(* PLC project TC3_TE1400_GeneratedModule_train_anarx_FB, Beckhoff Automation GmbH & Co. KG TwinCAT 3 Function - TE1400 1.2.1240 *)
(* stored: companyURL www.beckhoff.com, creationDateTime 2022-07-14T09:12:33 *)

TYPE E_TcMatSimDataAreaType : (NotSpecified := 0, Standard, InputSrc, InputDst, OutputSrc, OutputDst, InternalDa, MArea, RetainDa);
END_TYPE

TYPE ST_TcMatSimObjectDataAreaInfo : STRUCT
  pPlcVar : PVOID;
  pModuleProcImg : PVOID;
  nSize : UDINT;
  nDataAreaId : UDINT;
  eDataAreaType : E_TcMatSimDataAreaType;
END_STRUCT;
END_TYPE

{attribute 'pack_mode' := '4'}
TYPE ST_train_anarxInitData : STRUCT
  Header : TComInitDataHdr;
  CallByHdr : TComInitDataElmHdr;
  CallBy : TctModuleCallByType;
  ExecutionSequenceHdr : TComInitDataElmHdr;
  ExecutionSequence : TctModuleExecutionSequenceType;
  StepSizeHdr : TComInitDataElmHdr;
  StepSize : TctStepSizeType;
  ExtendedFileAccessOIDHdr : TComInitDataElmHdr;
  ExtendedFileAccessOID : OTCID;
  ExecuteModelCodeHdr : TComInitDataElmHdr;
  ExecuteModelCode : BOOL;
  ModelParametersHdr : TComInitDataElmHdr;
  ModelParameters : P_train_anarx_T;
  ContextInfoArr_0_TaskOidHdr : TComInitDataElmHdr;
  ContextInfoArr_0_TaskOid : OTCID;
  ContextInfoArr_0_TaskPriorityHdr : TComInitDataElmHdr;
  ContextInfoArr_0_TaskPriority : UDINT;
  ContextInfoArr_0_TaskCycleTimeNsHdr : TComInitDataElmHdr;
  ContextInfoArr_0_TaskCycleTimeNs : UDINT;
  ContextInfoArr_0_TaskPortHdr : TComInitDataElmHdr;
  ContextInfoArr_0_TaskPort : UINT;
  ContextInfoArr_0_TaskSortOrderHdr : TComInitDataElmHdr;
  ContextInfoArr_0_TaskSortOrder : UDINT;
END_STRUCT;
END_TYPE

TYPE ST_train_anarx_Input : STRUCT
  Position_Increments : UDINT;
  Velocity_Increments : LREAL;
  DMS : DINT;
  actual_torque : INT;
END_STRUCT;
END_TYPE

TYPE ST_train_anarx_Output : STRUCT
  Control_Word : UINT;
  Target_Torque : INT;
  trigger : USINT;
  StartMeasurement : BOOL;
END_STRUCT;
END_TYPE

FUNCTION_BLOCK FB_TcMatSimObject
  VAR_INPUT
    bWriteFbInputValues : BOOL := TRUE;  (* set this flag to write FB input values to the TcComObject's input DataAreas. This will overwrite the mapped input values before module execution. Set to FALSE to read the mapped input values from the TcComObject to the FB. *)
  END_VAR
  VAR
    pDataAreas : POINTER TO ST_TcMatSimObjectDataAreaInfo;  (* process image src and dst pointers and sizes *)
    nDataAreas : UDINT;
    ipObjSrv : ITComObjectServer;  (* global interface pointers *)
    ipTcComObj : ITComObject;  (* object interface pointers *)
    ipTcCyclic : ITcCyclic;
    ipTcPostCyclic : ITcPostCyclic;
    ipTcAdi : ITcADI;
    ipTask : ITcTask;  (* task interface pointers *)
    pInitData : POINTER TO TComInitDataHdr;  (* initial parameters *)
    hResult : HRESULT;  (* hResult of interface calls (0 if no error) *)
    moduleClsId : CLSID;  (* module class ID *)
    assignedClsId : CLSID;  (* expected/desired module class ID *)
    bClassIdVerified : BOOL;
    bDynInstance : BOOL;  (* flag indicating whether the module instance was created dynamically *)
    eInitialObjState : TCOM_STATE := TCOM_STATE.TCOM_STATE_INIT;  (* the object state at the time FB_init was called, FB_exit will try to switch to this state (only if this means to shift down) *)
  END_VAR

            
          

{attribute 'object_name' := 'ReleaseTcComInterface'}
METHOD ReleaseTcComInterface : HRESULT
  VAR
    nStateChangeCnt : DINT := 0;
  END_VAR
                  
IF (ipTcComObj<>0) THEN
  WHILE (State>eInitialObjState AND nStateChangeCnt<1000) DO
    State := eInitialObjState;
    nStateChangeCnt := nStateChangeCnt+1;
  END_WHILE
  ReleaseObjInterfaces();
  IF (bDynInstance) THEN
    ReleaseTcComInterface := TC3_MODULE.FW_ObjMgr_DeleteInstance(ADR(ipTcComObj));
  ELSE
    ipTcComObj.TcRelease();
  END_IF
  ipTcComObj := 0;
END_IF
                  
                
END_METHOD

{attribute 'object_name' := 'ReleaseObjInterfaces'}
METHOD ReleaseObjInterfaces : HRESULT
                  
// release interface pointers
IF (ipTcCyclic<>0) THEN
  ipTcCyclic.TcRelease();
  ipTcCyclic := 0;
END_IF
IF (ipTcPostCyclic<>0) THEN
  ipTcPostCyclic.TcRelease();
  ipTcPostCyclic := 0;
END_IF
IF (ipTcAdi<>0) THEN
  ipTcAdi.TcRelease();
  ipTcAdi := 0;
END_IF
                  
                
END_METHOD

{attribute 'object_name' := 'Internal_SetObjState'}
METHOD Internal_SetObjState
  VAR_INPUT
    hr : REFERENCE TO HRESULT;
    nextState : TCOM_STATE;
  END_VAR
                  
// verify class id
IF (SUCCEEDED(hr)) THEN
  hr := VerifyClassId();
END_IF

// switch object state
IF (SUCCEEDED(hr) AND nextState>=TCOM_STATE_INIT) THEN
  IF (ipTcComObj=0) THEN
    hr := Tc2_System.E_HRESULTAdsErr.NOINTERFACE;
  END_IF
  IF (ipObjSrv=0) THEN
    hr := Tc2_System.E_HRESULTAdsErr.NOINTERFACE;
  END_IF
  IF (SUCCEEDED(hr)) THEN
    hr := ipTcComObj.TcSetObjState(nextState,ipObjSrv,pInitData);
  END_IF
END_IF
                  
                
END_METHOD

{attribute 'object_name' := 'FB_init'}
METHOD FB_init : BOOL
  VAR_INPUT
    bInitRetains : BOOL;  (* init retain variables *)
    bInCopyCode : BOOL;  (* Online Change *)
    oid : OTCID;
  END_VAR
                  
FB_init := SUCCEEDED(Init(oid));
                  
                
END_METHOD

{attribute 'object_name' := 'GetObjPara'}
METHOD GetObjPara : HRESULT
  VAR_INPUT
    pid : PTCID;
    nData : UDINT;
    pData : PVOID;
  END_VAR
                  
IF (ipTcComObj=0) THEN
  GetObjPara := Tc2_System.E_HRESULTAdsErr.NOINTERFACE;
END_IF

IF (SUCCEEDED(GetObjPara)) THEN
  GetObjPara := ipTcComObj.TcGetObjPara(pid:=pid,nData,pData,0);
END_IF
                  
                
END_METHOD

{attribute 'object_name' := 'QueryObjInterface'}
METHOD QueryObjInterface
  VAR_INPUT
    hr : REFERENCE TO HRESULT;
    iid : REFERENCE TO IID;
    pipItf : POINTER TO ITcUnknown;
  END_VAR
  VAR CONSTANT
    pNull : PVOID := 0;
  END_VAR
                  
IF (SUCCEEDED(hr)) THEN
  IF (ipTcComObj=0) THEN
    hr := Tc2_System.E_HRESULTAdsErr.NOINTERFACE;
  ELSIF (pipItf^=ULINT_TO_DWORD(pNull)) THEN
    hr := ipTcComObj.TcQueryInterface(iid:= iid, pipItf:=pipItf);
  END_IF
END_IF
                  
                
END_METHOD

{attribute 'object_name' := 'SaveOnlineParametersForInit'}
METHOD SaveOnlineParametersForInit : HRESULT
  VAR
    idx : UINT;
    pInitElemHdr : POINTER TO TComInitDataElmHdr;
    pData : PVOID;
    nData : UDINT;
  END_VAR
  VAR CONSTANT
    nInitDataAlignment : UDINT := 4;
  END_VAR
                  IF (pInitData<>0) THEN
  pInitElemHdr := pInitData + SIZEOF(pInitData^);
  FOR idx:=1 TO pInitData^.uiElmCnt DO
    pData := pInitElemHdr + ULINT_TO_DWORD(SIZEOF(pInitElemHdr^));
    nData := pInitElemHdr^.cbData;
    SaveOnlineParametersForInit := GetObjPara(pInitElemHdr^.indexOffset,nData,pData);
    IF (FAILED(SaveOnlineParametersForInit)) THEN
      RETURN;
    END_IF
    pInitElemHdr := pData + (nInitDataAlignment*((nData + nInitDataAlignment - 1)/nInitDataAlignment));
  END_FOR
ELSE
	SaveOnlineParametersForInit := Tc2_System.E_HRESULTAdsErr.NOTINIT;
END_IF
                  
                
END_METHOD

{attribute 'object_name' := 'ResetHresult'}
METHOD ResetHresult
                  hResult := S_OK;
                
END_METHOD

{attribute 'object_name' := 'Execute'}
METHOD Execute : HRESULT
  VAR
    nDaIdx : UDINT;
    pCurDataArea : POINTER TO ST_TcMatSimObjectDataAreaInfo;
  END_VAR
                  
IF (SUCCEEDED(hResult)) THEN
  hResult := VerifyClassId();
END_IF

IF (SUCCEEDED(hResult) AND State<>TCOM_STATE_OP) THEN
  hResult := Tc2_System.E_HRESULTAdsErr.NOTREADY;
END_IF

// get image pointers
IF (SUCCEEDED(hResult)) THEN
  GetImagePtrs(hResult);
END_IF

// copy inputs
IF (pDataAreas<>0 AND nDataAreas>0 AND bWriteFbInputValues) THEN
  FOR nDaIdx:=0 TO nDataAreas-1 DO
    IF (FAILED(hResult))THEN
      CONTINUE;
    END_IF
    pCurDataArea := pDataAreas + nDaIdx*SIZEOF(ST_TcMatSimObjectDataAreaInfo);
    IF ((pCurDataArea^.eDataAreaType <> E_TcMatSimDataAreaType.InputDst))THEN
      CONTINUE;
    END_IF
    IF (pCurDataArea^.pModuleProcImg<>0 AND pCurDataArea^.pPlcVar<>0) THEN
      MEMCPY(pCurDataArea^.pModuleProcImg,pCurDataArea^.pPlcVar,pCurDataArea^.nSize);
    ELSE
      hResult := Tc2_System.E_HRESULTAdsErr.NOINTERFACE;
    END_IF
  END_FOR
END_IF

// call cycle update
IF (SUCCEEDED(hResult)) THEN
  IF (ipTcCyclic<>0) THEN
    hResult := ipTcCyclic.CycleUpdate(ipTask:= ipTask, ipCaller:= 0, context:= 0);
  ELSE
    hResult := Tc2_System.E_HRESULTAdsErr.NOINTERFACE;
  END_IF
END_IF

// copy outputs
IF (pDataAreas<>0 AND nDataAreas>0) THEN
  FOR nDaIdx:=0 TO nDataAreas-1 DO
    IF (FAILED(hResult))THEN
      CONTINUE;
    END_IF
    pCurDataArea := pDataAreas + nDaIdx*SIZEOF(ST_TcMatSimObjectDataAreaInfo);
    IF ((pCurDataArea^.eDataAreaType = E_TcMatSimDataAreaType.OutputSrc) OR NOT bWriteFbInputValues) THEN
      IF (pCurDataArea^.pModuleProcImg<>0 AND pCurDataArea^.pPlcVar<>0) THEN
        MEMCPY(pCurDataArea^.pPlcVar,pCurDataArea^.pModuleProcImg,pCurDataArea^.nSize);
      ELSE
        hResult := Tc2_System.E_HRESULTAdsErr.NOINTERFACE;
      END_IF
    END_IF
  END_FOR
END_IF


// call post cyclic update
IF (SUCCEEDED(hResult)) THEN
  IF (ipTcPostCyclic<>0) THEN
    hResult := ipTcPostCyclic.PostCyclicUpdate(ipTask:= 0, ipCaller:= 0, context:= 0);
  ELSE
    hResult := Tc2_System.E_HRESULTAdsErr.NOINTERFACE;
  END_IF
END_IF

ReleaseImagePtrs();

Execute := hResult;
                  
                
END_METHOD

{attribute 'object_name' := 'GetImagePtrs'}
METHOD GetImagePtrs
  VAR_INPUT
    hr : REFERENCE TO HRESULT;
  END_VAR
  VAR
    nDaIdx : UDINT;
    pCurDataArea : POINTER TO ST_TcMatSimObjectDataAreaInfo;
  END_VAR
                  
IF (ipTcAdi=0) THEN
  hr := Tc2_System.E_HRESULTAdsErr.NOINTERFACE;
END_IF
IF(State<>TCOM_STATE_OP)THEN
  hr := Tc2_System.E_HRESULTAdsErr.INVALIDSTATE;
END_IF


// get pointers to process images
IF (pDataAreas<>0 AND nDataAreas>0) THEN
  FOR nDaIdx:=0 TO nDataAreas-1 DO
    pCurDataArea := pDataAreas + nDaIdx*SIZEOF(ST_TcMatSimObjectDataAreaInfo);
    IF (FAILED(hr))THEN
      CONTINUE;
    END_IF
    IF ((pCurDataArea^.eDataAreaType <> E_TcMatSimDataAreaType.InputDst) AND (pCurDataArea^.eDataAreaType <> E_TcMatSimDataAreaType.OutputSrc))THEN
      CONTINUE;
    END_IF
    IF (pCurDataArea^.pModuleProcImg=0 AND pCurDataArea^.nSize>0) THEN
      hr := ipTcAdi.GetImagePtr(size:= pCurDataArea^.nSize , offs:=0 , adi_x:=pCurDataArea^.nDataAreaId , ppData:=ADR(pCurDataArea^.pModuleProcImg));
    END_IF
  END_FOR
END_IF

IF (FAILED(hr)) THEN
  ReleaseImagePtrs();
END_IF
                  
                
END_METHOD

{attribute 'object_name' := 'VerifyClassId'}
METHOD VerifyClassId : HRESULT
  VAR
    emptyClsId : CLSID;
  END_VAR
                  memset(ADR(emptyClsId),0,SIZEOF(emptyClsId));
IF (bClassIdVerified) THEN
  // class ID was already verified
  VerifyClassId := Tc2_System.E_HRESULTAdsErr.HRESULT_ADS_NOERROR;
ELSIF (memcmp(ADR(assignedClsId),ADR(emptyClsId),SIZEOF(assignedClsId))=0) THEN
  // skip class ID verification if no assignedClsId specified
  VerifyClassId := Tc2_System.E_HRESULTAdsErr.HRESULT_ADS_NOERROR;
ELSE
  // verify class ID
  VerifyClassId := ReadModuleClassId();

  IF (SUCCEEDED(VerifyClassId)) THEN
    IF (memcmp(ADR(assignedClsId),ADR(moduleClsId),SIZEOF(assignedClsId))<>0) THEN
     VerifyClassId := Tc2_System.E_HRESULTAdsErr.INVALIDCLSID;
    END_IF
  END_IF
  bClassIdVerified := SUCCEEDED(VerifyClassId);
END_IF
                  
                
END_METHOD

{attribute 'object_name' := 'SetObjPara'}
METHOD SetObjPara : HRESULT
  VAR_INPUT
    pid : PTCID;
    nData : UDINT;
    pData : PVOID;
  END_VAR
                  
IF (ipTcComObj=0) THEN
  SetObjPara := Tc2_System.E_HRESULTAdsErr.NOINTERFACE;
END_IF

IF (SUCCEEDED(SetObjPara)) THEN
  SetObjPara := ipTcComObj.TcSetObjPara(pid:=pid,nData,pData,0);
END_IF
                  
                
END_METHOD

{attribute 'object_name' := 'QueryTcComInterface'}
METHOD QueryTcComInterface
  VAR_INPUT
    hr : REFERENCE TO HRESULT;
    oid : OTCID;
  END_VAR
                  
IF (ipObjSrv=0) THEN
  hr := Tc2_System.E_HRESULTAdsErr.NOINTERFACE;
END_IF

IF (SUCCEEDED(hr) AND ipTcComObj=0) THEN
  bDynInstance := FALSE;
  IF(oid>0) THEN
    // query interface of existing object
    hr := ipObjSrv.TcQueryObjectInterface(oid,IID_ITComObject,ADR(ipTcComObj));
  ELSE
    // create new instance and get the object interface
    hr := ipObjSrv.TcCreateInstance(assignedClsId,IID_ITComObject,ADR(ipTcComObj));
    IF (SUCCEEDED(hr)) THEN
      bDynInstance := TRUE;
      hr := ipTcComObj.TcSetObjectId(OTCID_CreateNewId);
    END_IF
  END_IF
  IF (SUCCEEDED(hr)) THEN
    eInitialObjState := State;
  END_IF
END_IF
                  
                
END_METHOD

{attribute 'object_name' := 'ReleaseImagePtrs'}
METHOD ReleaseImagePtrs : HRESULT
  VAR
    nDaIdx : UDINT;
    pCurDataArea : POINTER TO ST_TcMatSimObjectDataAreaInfo;
  END_VAR
                  
IF (ipTcAdi=0) THEN
  ReleaseImagePtrs := Tc2_System.E_HRESULTAdsErr.NOINTERFACE;
END_IF

IF (SUCCEEDED(ReleaseImagePtrs) AND pDataAreas<>0 AND nDataAreas>0) THEN
  // release pointers to the simulink module process images
  FOR nDaIdx:=0 TO nDataAreas-1 DO
    pCurDataArea := pDataAreas + nDaIdx*SIZEOF(ST_TcMatSimObjectDataAreaInfo);

    IF (pCurDataArea^.pModuleProcImg<>0) THEN
      ipTcAdi.ReleaseImagePtr(pData:=pCurDataArea^.pModuleProcImg);
      pCurDataArea^.pModuleProcImg := 0;
    END_IF
  END_FOR
END_IF
                  
                
END_METHOD

{attribute 'object_name' := 'FB_exit'}
METHOD FB_exit : BOOL
  VAR_INPUT
    bInCopyCode : BOOL;  (* Online Change *)
  END_VAR
                  
IF (NOT bInCopyCode) THEN
  IF (ipObjSrv<>0) THEN
    ipObjSrv.TcRelease();
    ipObjSrv := 0;
  END_IF

  ReleaseTcComInterface();
END_IF
                  
                
END_METHOD

{attribute 'object_name' := 'InitObjName'}
METHOD InitObjName
  VAR_INPUT
    hr : REFERENCE TO HRESULT;
  END_VAR
  VAR
    objectName : STRING(255) := 'TcMatSimObject_PlcRtFbInstance';
    oid : OTCID;
  END_VAR
                  
IF (SUCCEEDED(hr)) THEN
  hr := ipTcComObj.TcGetObjectId(oid);
END_IF

IF (SUCCEEDED(hr) and bDynInstance) THEN
  objectName := TC2_STANDARD.CONCAT(objectName,'_');
  objectName := TC2_STANDARD.CONCAT(objectName,UDINT_TO_STRING(oid));
  hr := ipTcComObj.TcSetObjectName(ADR(objectName));
END_IF
                  
                
END_METHOD

{attribute 'object_name' := 'SetObjState'}
METHOD SetObjState : HRESULT
  VAR_INPUT
    finalState : TCOM_STATE;
  END_VAR
  VAR
    bShiftUp : BOOL;
    bShiftDown : BOOL;
    currentState : TCOM_STATE;
  END_VAR
                  
currentState := State;

bShiftUp := finalState>currentState;
bShiftDown := finalState<currentState;

// do not switch up on error
IF (FAILED(hresult)) THEN
  bShiftUp := FALSE;
END_IF
// reset existing error on switching down
IF (bShiftDown) THEN
  ResetHresult();
END_IF

// prepared state switch
CASE currentState OF
  TCOM_STATE_INIT:
    IF(bShiftUp) THEN
      QueryTcComInterface(hResult,0);
      Internal_SetObjState(hResult,TCOM_STATE.TCOM_STATE_PREOP);
      InitObjName(hResult);
    END_IF

  TCOM_STATE_PREOP:
    IF(bShiftUp) THEN
      Internal_SetObjState(hResult,TCOM_STATE.TCOM_STATE_SAFEOP);
      QueryObjInterfaces(hResult);
    ELSIF (bShiftDown) THEN
      Internal_SetObjState(hResult,TCOM_STATE.TCOM_STATE_INIT);
    END_IF

  TCOM_STATE_SAFEOP:
    IF(bShiftUp) THEN
      Internal_SetObjState(hResult,TCOM_STATE.TCOM_STATE_OP);
      QueryObjInterfaces(hResult);
    ELSIF (bShiftDown) THEN
      Internal_SetObjState(hResult,TCOM_STATE.TCOM_STATE_PREOP);
      ReleaseObjInterfaces();
    END_IF


  TCOM_STATE_OP:
    IF (bShiftDown) THEN
      Internal_SetObjState(hResult,TCOM_STATE.TCOM_STATE_SAFEOP);
    END_IF
END_CASE

SetObjState := hResult;
                  
                
END_METHOD

{attribute 'object_name' := 'QueryObjInterfaces'}
METHOD QueryObjInterfaces
  VAR_INPUT
    hr : REFERENCE TO HRESULT;
  END_VAR
                  
IF(State<TCOM_STATE_PREOP)THEN
  hr := Tc2_System.E_HRESULTAdsErr.INVALIDSTATE;
END_IF

//cyclic interface
QueryObjInterface(hr,IID_ITCCYCLIC,ADR(ipTcCyclic));
//post cyclic interface
QueryObjInterface(hr,IID_ITCPOSTCYCLIC,ADR(ipTcPostCyclic));
//adi interface
QueryObjInterface(hr,IID_ITcADI,ADR(ipTcAdi));
                  
                
END_METHOD

{attribute 'object_name' := 'Init'}
METHOD Init : HRESULT
  VAR_INPUT
    oid : OTCID;
  END_VAR
                  
// preinitialize variables
memset(ADR(moduleClsId),0,SIZEOF(moduleClsId));
bClassIdVerified := FALSE;
hResult := Tc2_System.E_HRESULTAdsErr.HRESULT_ADS_NOERROR;

// get object server
IF (ipObjSrv=0) THEN
  hResult := FW_ObjMgr_GetObjectServer(_AppInfo.ObjId,ADR(ipObjSrv));
END_IF

// try to get object interfaces
IF (SUCCEEDED(hresult)) THEN
  QueryTcComInterface(hResult,oid);
END_IF

// verify class id
IF (SUCCEEDED(hresult)) THEN
  hresult := VerifyClassId();
END_IF

// query interfaces, if the current state is higher than INIT
IF (SUCCEEDED(hresult) AND State>TCOM_STATE.TCOM_STATE_INIT) THEN
  QueryObjInterfaces(hResult);
END_IF

// return value
Init := hresult;
                  
                
END_METHOD

{attribute 'object_name' := 'ReadModuleClassId'}
METHOD ReadModuleClassId : HRESULT
  VAR
    emptyClsId : CLSID;
  END_VAR
                  memset(ADR(emptyClsId),0,SIZEOF(emptyClsId));
IF (memcmp(ADR(moduleClsId),ADR(emptyClsId),SIZEOF(moduleClsId))=0) THEN
  IF (ipTcComObj=0) THEN
    ReadModuleClassId := Tc2_System.E_HRESULTAdsErr.NOINTERFACE;
  END_IF

  //objectClsId := clsid;
  IF (SUCCEEDED(ReadModuleClassId)) THEN
    ReadModuleClassId := ipTcComObj.GetClassId(moduleClsId);
  END_IF
END_IF
                
END_METHOD

METHOD PUBLIC AssignClassId
VAR_INPUT
	clsId : CLSID;
END_VAR
                  assignedClsId := clsId;
bClassIdVerified := false;
                  
                
END_METHOD

PROPERTY Error : BOOL
GET
                    Error := FAILED(hResult);
                  
END_GET
END_PROPERTY

METHOD PUBLIC SetDataAreaInfo
VAR_INPUT
  pDataAreas: POINTER TO ST_TcMatSimObjectDataAreaInfo;
  nDataAreas: UDINT;
END_VAR
                  
THIS^.nDataAreas := nDataAreas;
THIS^.pDataAreas := pDataAreas;
                  
                
END_METHOD

METHOD PUBLIC SetInitDataInfo
VAR_INPUT
  pInitData : POINTER TO TComInitDataHdr;
END_VAR
                  this^.pInitData := pInitData;
                
END_METHOD

PROPERTY ClassId : CLSID
GET
                    hResult := ReadModuleClassId();
ClassId := moduleClsId;
                    
                  
END_GET
END_PROPERTY

PROPERTY State : TCOM_STATE
GET
  VAR
    hr : HRESULT := S_OK;
    eObjState : TCOM_STATE;
  END_VAR
                    
IF (ipTcComObj<>0) THEN
  hr := ipTcComObj.TcGetObjState(ADR(eObjState));
IF (FAILED(hr)) THEN
  eObjState := TCOM_STATE.TCOM_STATE_INIT;
END_IF
ELSE
  eObjState := TCOM_STATE.TCOM_STATE_INIT;
END_IF
State := eObjState;
                    
                  
END_GET
SET
                    SetObjState(State);
                  
END_SET
END_PROPERTY

PROPERTY ErrorCode : HRESULT
GET
                    ErrorCode := hResult;
                  
END_GET
END_PROPERTY
END_FUNCTION_BLOCK

{attribute 'TcDependOnClassFactory' := 'train_anarx'}
FUNCTION_BLOCK FB_train_anarx EXTENDS FB_TcMatSimObject
  VAR_INPUT
    stInput : ST_train_anarx_Input;
  END_VAR
  VAR_OUTPUT
    stOutput : ST_train_anarx_Output;
  END_VAR
  VAR
    stInitData : ST_train_anarxInitData;
    arrDataAreas : ARRAY[1..2] OF ST_TcMatSimObjectDataAreaInfo;
    bParametersVerified : BOOL;
  END_VAR

            
          

{attribute 'object_name' := 'Internal_SetObjState'}
METHOD Internal_SetObjState
  VAR_INPUT
    hr : REFERENCE TO HRESULT;
    nextState : TCOM_STATE;
  END_VAR
                  
// update pointer to InitData structure
SetInitDataInfo(ADR(stInitData));
// call base method
SUPER^.Internal_SetObjState(hr,nextState);
                  
                
END_METHOD

{attribute 'object_name' := 'SaveOnlineParametersForInit'}
METHOD SaveOnlineParametersForInit : HRESULT
  VAR
    idx : UINT;
    pInitElemHdr : POINTER TO TComInitDataElmHdr;
    pData : PVOID;
    nData : UDINT;
  END_VAR
  VAR CONSTANT
    nInitDataAlignment : UDINT := 4;
  END_VAR
                  
// update pointer to InitData structure
SetInitDataInfo(ADR(stInitData));
// call base method
SaveOnlineParametersForInit := SUPER^.SaveOnlineParametersForInit();
                  
                
END_METHOD

METHOD FB_init : BOOL
  VAR_INPUT
    bInitRetains : BOOL;  (* if TRUE, the retain variables are initialized (warm start / cold start) *)
    bInCopyCode : BOOL;  (* if TRUE, the instance afterwards gets moved into the copy code (online change) *)
    oid : OTCID;
  END_VAR
  VAR
    clsId : CLSID;
  END_VAR
                  
// initialize flags
bParametersVerified := false;
                    
// set module class id for compatibility check
clsId.Data1 := 16#ed2a66fb;
clsId.Data2 := 16#550e;
clsId.Data3 := 16#4b31;
clsId.Data4[0] := 16#b5;
clsId.Data4[1] := 16#1b;
clsId.Data4[2] := 16#1e;
clsId.Data4[3] := 16#91;
clsId.Data4[4] := 16#4f;
clsId.Data4[5] := 16#8f;
clsId.Data4[6] := 16#f7;
clsId.Data4[7] := 16#c0;

AssignClassId(clsId);
                    
// initialize InitData structure with default values              
stInitData.CallByHdr.indexGroup := 0;
stInitData.CallByHdr.indexOffset := 16#00000000;
stInitData.CallByHdr.cbData := SIZEOF(stInitData.CallBy);
stInitData.CallBy := TctModuleCallByType.CyclicTask;
stInitData.ExecutionSequenceHdr.indexGroup := 0;
stInitData.ExecutionSequenceHdr.indexOffset := 16#00000001;
stInitData.ExecutionSequenceHdr.cbData := SIZEOF(stInitData.ExecutionSequence);
stInitData.ExecutionSequence := TctModuleExecutionSequenceType.StateUpdateAfterOutputMapping;
stInitData.StepSizeHdr.indexGroup := 0;
stInitData.StepSizeHdr.indexOffset := 16#00000002;
stInitData.StepSizeHdr.cbData := SIZEOF(stInitData.StepSize);
stInitData.StepSize := TctStepSizeType.RequireMatchingTaskCycleTime;
stInitData.ExtendedFileAccessOIDHdr.indexGroup := 0;
stInitData.ExtendedFileAccessOIDHdr.indexOffset := 16#00000005;
stInitData.ExtendedFileAccessOIDHdr.cbData := SIZEOF(stInitData.ExtendedFileAccessOID);
stInitData.ExtendedFileAccessOID := 0;
stInitData.ExecuteModelCodeHdr.indexGroup := 0;
stInitData.ExecuteModelCodeHdr.indexOffset := 16#00000008;
stInitData.ExecuteModelCodeHdr.cbData := SIZEOF(stInitData.ExecuteModelCode);
stInitData.ExecuteModelCode := 1;
stInitData.ModelParametersHdr.indexGroup := 0;
stInitData.ModelParametersHdr.indexOffset := 16#83000000;
stInitData.ModelParametersHdr.cbData := SIZEOF(stInitData.ModelParameters);
stInitData.ModelParameters._R[0] := 0.10557324255439252;
stInitData.ModelParameters._R[1] := 0.37689728877712958;
stInitData.ModelParameters._R[2] := 0.82623132681154499;
stInitData.ModelParameters._R[3] := 0.80515070185744342;
stInitData.ModelParameters._R[4] := 0.28033408284883216;
stInitData.ModelParameters._R[5] := 0.20419454517375848;
stInitData.ModelParameters._R[6] := 0.29127318222485832;
stInitData.ModelParameters._R[7] := 0.25248459304526055;
stInitData.ModelParameters._R[8] := 0.85181877670829109;
stInitData.ModelParameters._R[9] := 0.26730813856504498;
stInitData.ModelParameters._R[10] := 0.85973341835764761;
stInitData.ModelParameters._R[11] := 0.48821150954772086;
stInitData.ModelParameters._R[12] := 0.66695764239898803;
stInitData.ModelParameters._R[13] := 0.76922255995861488;
stInitData.ModelParameters._R[14] := 0.45433723001590831;
stInitData.ModelParameters._R[15] := 0.36540629909774192;
stInitData.ModelParameters._R[16] := 0.18448083270146118;
stInitData.ModelParameters._R[17] := 0.70086782168457618;
stInitData.ModelParameters._R[18] := 0.76784685041686818;
stInitData.ModelParameters._R[19] := 0.56414679263598622;
stInitData.ModelParameters._R[20] := 0.58598712526380503;
stInitData.ModelParameters._R[21] := 0.61005066126219132;
stInitData.ModelParameters._R[22] := 0.19543577562249415;
stInitData.ModelParameters._R[23] := 0.64329142670086592;
stInitData.ModelParameters._R[24] := 0.58267310864706856;
stInitData.ModelParameters._R[25] := 0.79798332299322849;
stInitData.ModelParameters._R[26] := 0.33180383592093965;
stInitData.ModelParameters._R[27] := 0.98316309922904865;
stInitData.ModelParameters._R[28] := 0.61220339829755299;
stInitData.ModelParameters._R[29] := 0.37845979384680939;
stInitData.ModelParameters._R[30] := 0.26096574430972613;
stInitData.ModelParameters._R[31] := 0.98801891092854388;
stInitData.ModelParameters._R[32] := 0.88761571192799182;
stInitData.ModelParameters._R[33] := 0.49443727460454467;
stInitData.ModelParameters._R[34] := 0.96137766517165912;
stInitData.ModelParameters._R[35] := 0.75085204485352486;
stInitData.ModelParameters._R[36] := 0.66551284350087503;
stInitData.ModelParameters._R[37] := 0.56475841691778406;
stInitData.ModelParameters._R[38] := 0.67811270612970664;
stInitData.ModelParameters._R[39] := 0.73032933705708902;
stInitData.ModelParameters._R[40] := 0.9876927697421114;
stInitData.ModelParameters._R[41] := 0.17853778300790973;
stInitData.ModelParameters._R[42] := 0.2112881137503454;
stInitData.ModelParameters._R[43] := 0.22263422347063244;
stInitData.ModelParameters._R[44] := 0.22981152085528173;
stInitData.ModelParameters._R[45] := 0.58054172851801422;
stInitData.ModelParameters._R[46] := 0.13458174770618431;
stInitData.ModelParameters._R[47] := 0.41675382902513802;
stInitData.ModelParameters._R[48] := 0.37503426129121775;
stInitData.ModelParameters._R[49] := 0.61532742494748438;
stInitData.ModelParameters._R[50] := 0.58497592475358873;
stInitData.ModelParameters._R[51] := 0.57088276882443501;
stInitData.ModelParameters._R[52] := 0.83801882588390086;
stInitData.ModelParameters._R[53] := 0.46346631174006891;
stInitData.ModelParameters._R[54] := 0.95558082085154439;
stInitData.ModelParameters._R[55] := 0.35709928964954307;
stInitData.ModelParameters._R[56] := 0.29876036646169085;
stInitData.ModelParameters._R[57] := 0.48986379749351949;
stInitData.ModelParameters._R[58] := 0.24301356646415506;
stInitData.ModelParameters._R[59] := 0.56396401425412857;
stInitData.ModelParameters._R[60] := 0.28037514198911928;
stInitData.ModelParameters._R[61] := 0.30519349579670008;
stInitData.ModelParameters._R[62] := 0.24886260905900215;
stInitData.ModelParameters._R[63] := 0.5294540187906408;
stInitData.ModelParameters._R[64] := 0.53146096958643707;
stInitData.ModelParameters._R[65] := 0.34765305839671429;
stInitData.ModelParameters._R[66] := 0.15713547018740073;
stInitData.ModelParameters._R[67] := 0.82999914974606137;
stInitData.ModelParameters._R[68] := 0.34671381817231139;
stInitData.ModelParameters._R[69] := 0.11129442711906647;
stInitData.ModelParameters._R[70] := 0.12533045888018424;
stInitData.ModelParameters._R[71] := 0.32318971865563034;
stInitData.ModelParameters._R[72] := 0.62869755633878344;
stInitData.ModelParameters._R[73] := 0.69689944130345438;
stInitData.ModelParameters._R[74] := 0.10259475882910257;
stInitData.ModelParameters._R[75] := 0.504612921588942;
stInitData.ModelParameters._R[76] := 0.82405522325355751;
stInitData.ModelParameters._R[77] := 0.23426045233071416;
stInitData.ModelParameters._R[78] := 0.13659391696110607;
stInitData.ModelParameters._R[79] := 0.33620017245498535;
stInitData.ModelParameters._R[80] := 0.23888235575200314;
stInitData.ModelParameters._R[81] := 0.39016605800346627;
stInitData.ModelParameters._R[82] := 0.61276603447948219;
stInitData.ModelParameters._R[83] := 0.2579770782045353;
stInitData.ModelParameters._R[84] := 0.8771624518519725;
stInitData.ModelParameters._R[85] := 0.55326589403810822;
stInitData.ModelParameters._R[86] := 0.58235210422493999;
stInitData.ModelParameters._R[87] := 0.98154545152029393;
stInitData.ModelParameters._R[88] := 0.83659615038432578;
stInitData.ModelParameters._R[89] := 0.79108937534487012;
stInitData.ModelParameters._R[90] := 0.29559361351651137;
stInitData.ModelParameters._R[91] := 0.11293767053593151;
stInitData.ModelParameters._R[92] := 0.21914052047882826;
stInitData.ModelParameters._R[93] := 0.82728419501927575;
stInitData.ModelParameters._R[94] := 0.59745588403726657;
stInitData.ModelParameters._R[95] := 0.99670425034860854;
stInitData.ModelParameters._R[96] := 0.21685275427583112;
stInitData.ModelParameters._R[97] := 0.9011734797642712;
stInitData.ModelParameters._R[98] := 0.32369112046493842;
stInitData.ModelParameters._R[99] := 0.71274938125352805;
stInitData.ModelParameters._R[100] := 0.1310510429654313;
stInitData.ModelParameters._R[101] := 0.4383330605382717;
stInitData.ModelParameters._R[102] := 0.30654446301433158;
stInitData.ModelParameters._R[103] := 0.87532334771214859;
stInitData.ModelParameters._R[104] := 0.7881416038506498;
stInitData.ModelParameters._R[105] := 0.29903673909793793;
stInitData.ModelParameters._R[106] := 0.18054953338168706;
stInitData.ModelParameters._R[107] := 0.35150006801524025;
stInitData.ModelParameters._R[108] := 0.60763011260701494;
stInitData.ModelParameters._R[109] := 0.67219780348968328;
stInitData.ModelParameters._R[110] := 0.21141218469813255;
stInitData.ModelParameters._R[111] := 0.23363444264258038;
stInitData.ModelParameters._R[112] := 0.95502425889513465;
stInitData.ModelParameters._R[113] := 0.67225964014063233;
stInitData.ModelParameters._R[114] := 0.61388033793257857;
stInitData.ModelParameters._R[115] := 0.54461364348051289;
stInitData.ModelParameters._R[116] := 0.7805403467686951;
stInitData.ModelParameters._R[117] := 0.25660513809200713;
stInitData.ModelParameters._R[118] := 0.98519948753497311;
stInitData.ModelParameters._R[119] := 0.12788370673330821;
stInitData.ModelParameters._R[120] := 0.38672759993250005;
stInitData.ModelParameters._R[121] := 0.67556889810283993;
stInitData.ModelParameters._R[122] := 0.81168147877462926;
stInitData.ModelParameters._R[123] := 0.46397047010591841;
stInitData.ModelParameters._R[124] := 0.28986124970741606;
stInitData.ModelParameters._R[125] := 0.17258139902247982;
stInitData.ModelParameters._R[126] := 0.61307238317924628;
stInitData.ModelParameters._R[127] := 0.89188121258164366;
stInitData.ModelParameters._R[128] := 0.30043225657821432;
stInitData.ModelParameters._R[129] := 0.71601528243326629;
stInitData.ModelParameters._R[130] := 0.90868555409275353;
stInitData.ModelParameters._R[131] := 0.53716709007367125;
stInitData.ModelParameters._R[132] := 0.42082395133622919;
stInitData.ModelParameters._R[133] := 0.16718964639417333;
stInitData.ModelParameters._R[134] := 0.75895365392615877;
stInitData.ModelParameters._R[135] := 0.67185678678085969;
stInitData.ModelParameters._R[136] := 0.88796076162712378;
stInitData.ModelParameters._R[137] := 0.62303474774669099;
stInitData.ModelParameters._R[138] := 0.42941298918691306;
stInitData.ModelParameters._R[139] := 0.99825181307434274;
stInitData.ModelParameters._R[140] := 0.37335410586877282;
stInitData.ModelParameters._R[141] := 0.23803968992299129;
stInitData.ModelParameters._R[142] := 0.9477463055419495;
stInitData.ModelParameters._R[143] := 0.78712318037915641;
stInitData.ModelParameters._R[144] := 0.47221674089303645;
stInitData.ModelParameters._R[145] := 0.5334175165756454;
stInitData.ModelParameters._R[146] := 0.20563370198365669;
stInitData.ModelParameters._R[147] := 0.23533219590845497;
stInitData.ModelParameters._R[148] := 0.76214597490525093;
stInitData.ModelParameters._R[149] := 0.30344628425015818;
stInitData.ModelParameters._R[150] := 0.7461972828186253;
stInitData.ModelParameters._R[151] := 0.70845951254033057;
stInitData.ModelParameters._R[152] := 0.11570620260467901;
stInitData.ModelParameters._R[153] := 0.13348175659892725;
stInitData.ModelParameters._R[154] := 0.51343849188399349;
stInitData.ModelParameters._R[155] := 0.6346454920872594;
stInitData.ModelParameters._R[156] := 0.76390258469096028;
stInitData.ModelParameters._R[157] := 0.71479891807934126;
stInitData.ModelParameters._R[158] := 0.8520955329408032;
stInitData.ModelParameters._R[159] := 0.36774770605365947;
stInitData.ModelParameters._R[160] := 0.68527294305296671;
stInitData.ModelParameters._R[161] := 0.75825763605206364;
stInitData.ModelParameters._R[162] := 0.442492312320236;
stInitData.ModelParameters._R[163] := 0.26523660922511622;
stInitData.ModelParameters._R[164] := 0.92611249773951621;
stInitData.ModelParameters._R[165] := 0.99624815670176925;
stInitData.ModelParameters._R[166] := 0.83860835530852751;
stInitData.ModelParameters._R[167] := 0.16379166188501976;
stInitData.ModelParameters._R[168] := 0.33580058998178808;
stInitData.ModelParameters._R[169] := 0.1264089858879642;
stInitData.ModelParameters._R[170] := 0.72140763008226205;
stInitData.ModelParameters._R[171] := 0.34798352409116884;
stInitData.ModelParameters._R[172] := 0.640715985720549;
stInitData.ModelParameters._R[173] := 0.2937509076499365;
stInitData.ModelParameters._R[174] := 0.89480038722921906;
stInitData.ModelParameters._R[175] := 0.30498145409302474;
stInitData.ModelParameters._R[176] := 0.18162286441150155;
stInitData.ModelParameters._R[177] := 0.27939606853906462;
stInitData.ModelParameters._R[178] := 0.93524197073824922;
stInitData.ModelParameters._R[179] := 0.46795873890621653;
stInitData.ModelParameters._R[180] := 0.3657039093014387;
stInitData.ModelParameters._R[181] := 0.22707155749850741;
stInitData.ModelParameters._R[182] := 0.27259830118886458;
stInitData.ModelParameters._R[183] := 0.30659519459390916;
stInitData.ModelParameters._R[184] := 0.54447792689419161;
stInitData.ModelParameters._R[185] := 0.29777571094884292;
stInitData.ModelParameters._R[186] := 0.39413566912408837;
stInitData.ModelParameters._R[187] := 0.93593064353318722;
stInitData.ModelParameters._R[188] := 0.49635429830703071;
stInitData.ModelParameters._R[189] := 0.92973934292780613;
stInitData.ModelParameters._R[190] := 0.42456882458900169;
stInitData.ModelParameters._R[191] := 0.80976278058629991;
stInitData.ModelParameters._R[192] := 0.21068401684477067;
stInitData.ModelParameters._R[193] := 0.44790493063539816;
stInitData.ModelParameters._R[194] := 0.99090963182905234;
stInitData.ModelParameters._R[195] := 0.29135520463117359;
stInitData.ModelParameters._R[196] := 0.83991877173611729;
stInitData.ModelParameters._R[197] := 0.62809024129315394;
stInitData.ModelParameters._R[198] := 0.25474376882492666;
stInitData.ModelParameters._R[199] := 0.2249620465499598;
stInitData.ModelParameters._R[200] := 0.88341441934848441;
stInitData.ModelParameters._R[201] := 0.58577012038900855;
stInitData.ModelParameters._R[202] := 0.33090995268843726;
stInitData.ModelParameters._R[203] := 0.66091741724418596;
stInitData.ModelParameters._R[204] := 0.55189977212552177;
stInitData.ModelParameters._R[205] := 0.86236996888840178;
stInitData.ModelParameters._R[206] := 0.42056115860986709;
stInitData.ModelParameters._R[207] := 0.57663287073034863;
stInitData.ModelParameters._R[208] := 0.41407613186463088;
stInitData.ModelParameters._R[209] := 0.66369799858103751;
stInitData.ModelParameters._R[210] := 0.73397447895275769;
stInitData.ModelParameters._R[211] := 0.84560850894207618;
stInitData.ModelParameters._R[212] := 0.1543484491420333;
stInitData.ModelParameters._R[213] := 0.42034593324311131;
stInitData.ModelParameters._R[214] := 0.58793050066342456;
stInitData.ModelParameters._R[215] := 0.38726271048322591;
stInitData.ModelParameters._R[216] := 0.82891526818947137;
stInitData.ModelParameters._R[217] := 0.75891955962047508;
stInitData.ModelParameters._R[218] := 0.12415351336074848;
stInitData.ModelParameters._R[219] := 0.88932413702636026;
stInitData.ModelParameters._R[220] := 0.78501003919158308;
stInitData.ModelParameters._R[221] := 0.87887990034886043;
stInitData.ModelParameters._R[222] := 0.31458755280054029;
stInitData.ModelParameters._R[223] := 0.89830256244181073;
stInitData.ModelParameters._R[224] := 0.93307822833921561;
stInitData.ModelParameters._R[225] := 0.67770559628803595;
stInitData.ModelParameters._R[226] := 0.72446572977946699;
stInitData.ModelParameters._R[227] := 0.25602043805088243;
stInitData.ModelParameters._R[228] := 0.24794536190901026;
stInitData.ModelParameters._R[229] := 0.85146001476637878;
stInitData.ModelParameters._R[230] := 0.57313340411414349;
stInitData.ModelParameters._R[231] := 0.32304869289507421;
stInitData.ModelParameters._R[232] := 0.41567914109382975;
stInitData.ModelParameters._R[233] := 0.51139670927512992;
stInitData.ModelParameters._R[234] := 0.66770088401566596;
stInitData.ModelParameters._R[235] := 0.82589630948387716;
stInitData.ModelParameters._R[236] := 0.16291924961090168;
stInitData.ModelParameters._R[237] := 0.54957861741194936;
stInitData.ModelParameters._R[238] := 0.29813706471814461;
stInitData.ModelParameters._R[239] := 0.63583548083331809;
stInitData.ModelParameters._R[240] := 0.90775741934187315;
stInitData.ModelParameters._R[241] := 0.86766773527079433;
stInitData.ModelParameters._R[242] := 0.60922014661752977;
stInitData.ModelParameters._R[243] := 0.36539394454003538;
stInitData.ModelParameters._R[244] := 0.81334168852802424;
stInitData.ModelParameters._R[245] := 0.26269387590690702;
stInitData.ModelParameters._R[246] := 0.90362203266825714;
stInitData.ModelParameters._R[247] := 0.63554774727020691;
stInitData.ModelParameters._R[248] := 0.81714898754820031;
stInitData.ModelParameters._R[249] := 0.38689426415564299;
stInitData.ModelParameters._R[250] := 0.19867873837003591;
stInitData.ModelParameters._R[251] := 0.86502678641193853;
stInitData.ModelParameters._R[252] := 0.69156859731176812;
stInitData.ModelParameters._R[253] := 0.16764519909088638;
stInitData.ModelParameters._R[254] := 0.98370153501708402;
stInitData.ModelParameters._R[255] := 0.77492790018026447;
stInitData.ModelParameters._R[256] := 0.44603637933589013;
stInitData.ModelParameters._R[257] := 0.21472382368026849;
stInitData.ModelParameters._R[258] := 0.3615512419311373;
stInitData.ModelParameters._R[259] := 0.20007592368854937;
stInitData.ModelParameters._R[260] := 0.1470573042325386;
stInitData.ModelParameters._R[261] := 0.29038242952094107;
stInitData.ModelParameters._R[262] := 0.37499319372845596;
stInitData.ModelParameters._R[263] := 0.47612551659678559;
stInitData.ModelParameters._R[264] := 0.66186100168855111;
stInitData.ModelParameters._R[265] := 0.26251152551092138;
stInitData.ModelParameters._R[266] := 0.53911364663138861;
stInitData.ModelParameters._R[267] := 0.23403882063429615;
stInitData.ModelParameters._R[268] := 0.8736170242927358;
stInitData.ModelParameters._R[269] := 0.10409132378582837;
stInitData.ModelParameters._R[270] := 0.34487562128687926;
stInitData.ModelParameters._R[271] := 0.27086229551577223;
stInitData.ModelParameters._R[272] := 0.85423251602347439;
stInitData.ModelParameters._R[273] := 0.94067846218981321;
stInitData.ModelParameters._R[274] := 0.78289975211357121;
stInitData.ModelParameters._R[275] := 0.69332195830344101;
stInitData.ModelParameters._R[276] := 0.32629131492264263;
stInitData.ModelParameters._R[277] := 0.44576540003744813;
stInitData.ModelParameters._R[278] := 0.98718540165049029;
stInitData.ModelParameters._R[279] := 0.11961567189792122;
stInitData.ModelParameters._R[280] := 0.10540790812123817;
stInitData.ModelParameters._R[281] := 0.91637616055866067;
stInitData.ModelParameters._R[282] := 0.95197189511234326;
stInitData.ModelParameters._R[283] := 0.84859967918710844;
stInitData.ModelParameters._R[284] := 0.60787538798962948;
stInitData.ModelParameters._R[285] := 0.74051253740817069;
stInitData.ModelParameters._R[286] := 0.23127710025176662;
stInitData.ModelParameters._R[287] := 0.93485880319876535;
stInitData.ModelParameters._R[288] := 0.29984338297023116;
stInitData.ModelParameters._R[289] := 0.64541244320868685;
stInitData.ModelParameters._R[290] := 0.3359853236433189;
stInitData.ModelParameters._R[291] := 0.57651911847040904;
stInitData.ModelParameters._R[292] := 0.91983121884614039;
stInitData.ModelParameters._R[293] := 0.77636987482284803;
stInitData.ModelParameters._R[294] := 0.50138277656777952;
stInitData.ModelParameters._R[295] := 0.24451009809648941;
stInitData.ModelParameters._R[296] := 0.54112797363116483;
stInitData.ModelParameters._R[297] := 0.53365689643582459;
stInitData.ModelParameters._R[298] := 0.63073394821720952;
stInitData.ModelParameters._R[299] := 0.71320616839046835;
stInitData.ModelParameters._R[300] := 0.152781366398133;
stInitData.ModelParameters._R[301] := 0.24988598600219311;
stInitData.ModelParameters._R[302] := 0.91234320023084092;
stInitData.ModelParameters._R[303] := 0.73766185245344817;
stInitData.ModelParameters._R[304] := 0.62152472063085129;
stInitData.ModelParameters._R[305] := 0.749010842735361;
stInitData.ModelParameters._R[306] := 0.36734282545880059;
stInitData.ModelParameters._R[307] := 0.46668002635069061;
stInitData.ModelParameters._R[308] := 0.59397771619270534;
stInitData.ModelParameters._R[309] := 0.73524305426552117;
stInitData.ModelParameters._R[310] := 0.86897256747568863;
stInitData.ModelParameters._R[311] := 0.62636005761996572;
stInitData.ModelParameters._R[312] := 0.12517547152272973;
stInitData.ModelParameters._R[313] := 0.24900440964101156;
stInitData.ModelParameters._R[314] := 0.38531621638293445;
stInitData.ModelParameters._R[315] := 0.32068439406479421;
stInitData.ModelParameters._R[316] := 0.35116619008582051;
stInitData.ModelParameters._R[317] := 0.87150610792338112;
stInitData.ModelParameters._R[318] := 0.1216940424663239;
stInitData.ModelParameters._R[319] := 0.95880280796555961;
stInitData.ModelParameters._R[320] := 0.41315222867800305;
stInitData.ModelParameters._R[321] := 0.8913230267547817;
stInitData.ModelParameters._R[322] := 0.67891698926997557;
stInitData.ModelParameters._R[323] := 0.83581253490315921;
stInitData.ModelParameters._R[324] := 0.22903957947114192;
stInitData.ModelParameters._R[325] := 0.80574035080046913;
stInitData.ModelParameters._R[326] := 0.35726585547478107;
stInitData.ModelParameters._R[327] := 0.17225076941540352;
stInitData.ModelParameters._R[328] := 0.14739401725027385;
stInitData.ModelParameters._R[329] := 0.11279893764620889;
stInitData.ModelParameters._R[330] := 0.68954835598151598;
stInitData.ModelParameters._R[331] := 0.22053213943371852;
stInitData.ModelParameters._R[332] := 0.64842451092410858;
stInitData.ModelParameters._R[333] := 0.60198589242851619;
stInitData.ModelParameters._R[334] := 0.45368955279763212;
stInitData.ModelParameters._R[335] := 0.68651579020798248;
stInitData.ModelParameters._R[336] := 0.71742927880275587;
stInitData.ModelParameters._R[337] := 0.94693626739170522;
stInitData.ModelParameters._R[338] := 0.15349302930224087;
stInitData.ModelParameters._R[339] := 0.38438381201296357;
stInitData.ModelParameters._R[340] := 0.72674059072822905;
stInitData.ModelParameters._R[341] := 0.1496594826880803;
stInitData.ModelParameters._R[342] := 0.50801264343243691;
stInitData.ModelParameters._R[343] := 0.80321214852030343;
stInitData.ModelParameters._R[344] := 0.73917551242977952;
stInitData.ModelParameters._R[345] := 0.29922912677194707;
stInitData.ModelParameters._R[346] := 0.19259086267793316;
stInitData.ModelParameters._R[347] := 0.56950152767461293;
stInitData.ModelParameters._R[348] := 0.68013259859509967;
stInitData.ModelParameters._R[349] := 0.32267163539839483;
stInitData.ModelParameters._R[350] := 0.12135743063387079;
stInitData.ModelParameters._R[351] := 0.12163074679522888;
stInitData.ModelParameters._R[352] := 0.66437088527749222;
stInitData.ModelParameters._R[353] := 0.83526342519887209;
stInitData.ModelParameters._R[354] := 0.19978914631775679;
stInitData.ModelParameters._R[355] := 0.43145611507254178;
stInitData.ModelParameters._R[356] := 0.6627657885328494;
stInitData.ModelParameters._R[357] := 0.79916808761051239;
stInitData.ModelParameters._R[358] := 0.24841470716673836;
stInitData.ModelParameters._R[359] := 0.91956613789327468;
stInitData.ModelParameters._R[360] := 0.26368505905654394;
stInitData.ModelParameters._R[361] := 0.20887421507655551;
stInitData.ModelParameters._R[362] := 0.36627775148601416;
stInitData.ModelParameters._R[363] := 0.45812277250595557;
stInitData.ModelParameters._R[364] := 0.31932478395790986;
stInitData.ModelParameters._R[365] := 0.9559680907189928;
stInitData.ModelParameters._R[366] := 0.77707535653345561;
stInitData.ModelParameters._R[367] := 0.46541444629582718;
stInitData.ModelParameters._R[368] := 0.45581763060834479;
stInitData.ModelParameters._R[369] := 0.31517720633405094;
stInitData.ModelParameters._R[370] := 0.80949897839652796;
stInitData.ModelParameters._R[371] := 0.69621345837157977;
stInitData.ModelParameters._R[372] := 0.15412590646511184;
stInitData.ModelParameters._R[373] := 0.58591713594947004;
stInitData.ModelParameters._R[374] := 0.46331497675559208;
stInitData.ModelParameters._R[375] := 0.814884437583271;
stInitData.ModelParameters._R[376] := 0.13387222723219155;
stInitData.ModelParameters._R[377] := 0.60146680448763212;
stInitData.ModelParameters._R[378] := 0.82445152827733315;
stInitData.ModelParameters._R[379] := 0.54348906834022159;
stInitData.ModelParameters._R[380] := 0.69269713411288358;
stInitData.ModelParameters._R[381] := 0.25514753659702316;
stInitData.ModelParameters._R[382] := 0.10560804134717576;
stInitData.ModelParameters._R[383] := 0.39153831827923657;
stInitData.ModelParameters._R[384] := 0.42523969183533072;
stInitData.ModelParameters._R[385] := 0.59643829475383547;
stInitData.ModelParameters._R[386] := 0.82554392538697596;
stInitData.ModelParameters._R[387] := 0.29618124399879642;
stInitData.ModelParameters._R[388] := 0.20907371564641325;
stInitData.ModelParameters._R[389] := 0.13781450045128973;
stInitData.ModelParameters._R[390] := 0.47034172365320925;
stInitData.ModelParameters._R[391] := 0.98700157056170745;
stInitData.ModelParameters._R[392] := 0.29645947469739686;
stInitData.ModelParameters._R[393] := 0.44792143343658142;
stInitData.ModelParameters._R[394] := 0.54843768063649967;
stInitData.ModelParameters._R[395] := 0.97814847420911655;
stInitData.ModelParameters._R[396] := 0.21530688781650881;
stInitData.ModelParameters._R[397] := 0.24314115084623122;
stInitData.ModelParameters._R[398] := 0.73843607660435295;
stInitData.ModelParameters._R[399] := 0.70610392397078026;
stInitData.ModelParameters._R[400] := 0.23443766234740526;
stInitData.ModelParameters._R[401] := 0.28686849926681746;
stInitData.ModelParameters._R[402] := 0.31647415585882488;
stInitData.ModelParameters._R[403] := 0.70822749280565211;
stInitData.ModelParameters._R[404] := 0.90142253898236235;
stInitData.ModelParameters._R[405] := 0.82812183804419959;
stInitData.ModelParameters._R[406] := 0.71646289667170771;
stInitData.ModelParameters._R[407] := 0.43634551464021265;
stInitData.ModelParameters._R[408] := 0.11028856536443793;
stInitData.ModelParameters._R[409] := 0.46714177924020417;
stInitData.ModelParameters._R[410] := 0.94612785174578762;
stInitData.ModelParameters._R[411] := 0.43511679984160434;
stInitData.ModelParameters._R[412] := 0.20605936050945545;
stInitData.ModelParameters._R[413] := 0.67348460756901607;
stInitData.ModelParameters._R[414] := 0.96230253843573288;
stInitData.ModelParameters._R[415] := 0.35814750242233773;
stInitData.ModelParameters._R[416] := 0.32917259685697281;
stInitData.ModelParameters._R[417] := 0.94726133578403904;
stInitData.ModelParameters._R[418] := 0.67908353034157631;
stInitData.ModelParameters._R[419] := 0.33493270207602621;
stInitData.ModelParameters._R[420] := 0.19243937832619046;
stInitData.ModelParameters._R[421] := 0.47748006303902879;
stInitData.ModelParameters._R[422] := 0.65535783469451969;
stInitData.ModelParameters._R[423] := 0.69278849145054078;
stInitData.ModelParameters._R[424] := 0.5317368227387248;
stInitData.ModelParameters._R[425] := 0.76663965566094039;
stInitData.ModelParameters._R[426] := 0.46640329341501396;
stInitData.ModelParameters._R[427] := 0.41825103375716033;
stInitData.ModelParameters._R[428] := 0.72711909841220146;
stInitData.ModelParameters._R[429] := 0.67905595430868659;
stInitData.ModelParameters._R[430] := 0.56719652602572146;
stInitData.ModelParameters._R[431] := 0.75250946589571777;
stInitData.ModelParameters._R[432] := 0.78719884902238024;
stInitData.ModelParameters._R[433] := 0.47148791814140723;
stInitData.ModelParameters._R[434] := 0.66723464873266536;
stInitData.ModelParameters._R[435] := 0.50129522081835154;
stInitData.ModelParameters._R[436] := 0.41059096195532052;
stInitData.ModelParameters._R[437] := 0.69634460542605559;
stInitData.ModelParameters._R[438] := 0.78989497414276821;
stInitData.ModelParameters._R[439] := 0.98767963235270939;
stInitData.ModelParameters._R[440] := 0.10678434241318679;
stInitData.ModelParameters._R[441] := 0.70592521812539466;
stInitData.ModelParameters._R[442] := 0.21637896086290437;
stInitData.ModelParameters._R[443] := 0.81184604041400343;
stInitData.ModelParameters._R[444] := 0.86641736239962575;
stInitData.ModelParameters._R[445] := 0.77547261391326694;
stInitData.ModelParameters._R[446] := 0.73677542667582518;
stInitData.ModelParameters._R[447] := 0.68667236623162664;
stInitData.ModelParameters._R[448] := 0.95554493256201489;
stInitData.ModelParameters._R[449] := 0.24577315967153915;
stInitData.ModelParameters._R[450] := 0.82866702524621916;
stInitData.ModelParameters._R[451] := 0.23528913528247475;
stInitData.ModelParameters._R[452] := 0.14997863094262642;
stInitData.ModelParameters._R[453] := 0.54198128906490184;
stInitData.ModelParameters._R[454] := 0.79648881233112268;
stInitData.ModelParameters._R[455] := 0.11635958312044649;
stInitData.ModelParameters._R[456] := 0.92259447869078592;
stInitData.ModelParameters._R[457] := 0.63681822641280761;
stInitData.ModelParameters._R[458] := 0.92647284846823841;
stInitData.ModelParameters._R[459] := 0.97336185804999065;
stInitData.ModelParameters._R[460] := 0.21529527381400831;
stInitData.ModelParameters._R[461] := 0.88314464658754699;
stInitData.ModelParameters._R[462] := 0.73863955096073497;
stInitData.ModelParameters._R[463] := 0.50347420725913583;
stInitData.ModelParameters._R[464] := 0.3613179538285608;
stInitData.ModelParameters._R[465] := 0.69252420522469282;
stInitData.ModelParameters._R[466] := 0.54458641921381479;
stInitData.ModelParameters._R[467] := 0.20409850349150183;
stInitData.ModelParameters._R[468] := 0.69256055931806071;
stInitData.ModelParameters._R[469] := 0.15429867103657041;
stInitData.ModelParameters._R[470] := 0.18349912936828533;
stInitData.ModelParameters._R[471] := 0.31661178655057459;
stInitData.ModelParameters._R[472] := 0.77392877621886036;
stInitData.ModelParameters._R[473] := 0.92993788650001508;
stInitData.ModelParameters._R[474] := 0.39583467269852191;
stInitData.ModelParameters._R[475] := 0.24271753948384542;
stInitData.ModelParameters._R[476] := 0.19637295819771194;
stInitData.ModelParameters._R[477] := 0.86843749801439762;
stInitData.ModelParameters._R[478] := 0.27449892119745145;
stInitData.ModelParameters._R[479] := 0.55950124655645106;
stInitData.ModelParameters._R[480] := 0.53915774672632455;
stInitData.ModelParameters._R[481] := 0.51599295998428141;
stInitData.ModelParameters._R[482] := 0.69298303608109291;
stInitData.ModelParameters._R[483] := 0.38222494142028773;
stInitData.ModelParameters._R[484] := 0.72515382838467946;
stInitData.ModelParameters._R[485] := 0.51492978198192341;
stInitData.ModelParameters._R[486] := 0.89161056125575089;
stInitData.ModelParameters._R[487] := 0.7012967427413298;
stInitData.ModelParameters._R[488] := 0.33184366366116869;
stInitData.ModelParameters._R[489] := 0.99138501211896279;
stInitData.ModelParameters._R[490] := 0.55401597160654015;
stInitData.ModelParameters._R[491] := 0.60805639350437801;
stInitData.ModelParameters._R[492] := 0.56881106292144834;
stInitData.ModelParameters._R[493] := 0.32949877549311524;
stInitData.ModelParameters._R[494] := 0.44353311894120417;
stInitData.ModelParameters._R[495] := 0.81008268299689823;
stInitData.ModelParameters._R[496] := 0.85308100270603082;
stInitData.ModelParameters._R[497] := 0.78906587650562654;
stInitData.ModelParameters._R[498] := 0.62791302965107398;
stInitData.ModelParameters._R[499] := 0.67632007660311644;
stInitData.ModelParameters._R[500] := 0.34030408091641728;
stInitData.ModelParameters._R[501] := 0.71591502371925253;
stInitData.ModelParameters._R[502] := 0.92348050250032643;
stInitData.ModelParameters._R[503] := 0.6336184422769584;
stInitData.ModelParameters._R[504] := 0.83349727558941167;
stInitData.ModelParameters._R[505] := 0.11621515424988069;
stInitData.ModelParameters._R[506] := 0.63264035902434101;
stInitData.ModelParameters._R[507] := 0.30708641022712674;
stInitData.ModelParameters._R[508] := 0.69246503778722046;
stInitData.ModelParameters._R[509] := 0.8866863640399919;
stInitData.ModelParameters._R[510] := 0.80138578477839517;
stInitData.ModelParameters._R[511] := 0.37291299516100718;
stInitData.ModelParameters._R[512] := 0.27350690652011866;
stInitData.ModelParameters._R[513] := 0.57041975064277073;
stInitData.ModelParameters._R[514] := 0.52684748062644526;
stInitData.ModelParameters._R[515] := 0.29922282355750979;
stInitData.ModelParameters._R[516] := 0.41415936410911525;
stInitData.ModelParameters._R[517] := 0.20305408105851458;
stInitData.ModelParameters._R[518] := 0.90519022810465244;
stInitData.ModelParameters._R[519] := 0.13917400381191752;
stInitData.ModelParameters._R[520] := 0.79885942042333791;
stInitData.ModelParameters._R[521] := 0.47511965113700749;
stInitData.ModelParameters._R[522] := 0.99212645040435821;
stInitData.ModelParameters._R[523] := 0.36810467761914256;
stInitData.ModelParameters._R[524] := 0.96066888548751384;
stInitData.ModelParameters._R[525] := 0.90804498394638178;
stInitData.ModelParameters._R[526] := 0.34708707280274925;
stInitData.ModelParameters._R[527] := 0.82824457799393036;
stInitData.ModelParameters._R[528] := 0.40907312882331792;
stInitData.ModelParameters._R[529] := 0.64138469990633729;
stInitData.ModelParameters._R[530] := 0.28727045087306335;
stInitData.ModelParameters._R[531] := 0.47055639864853438;
stInitData.ModelParameters._R[532] := 0.63570172165863159;
stInitData.ModelParameters._R[533] := 0.16775374466707763;
stInitData.ModelParameters._R[534] := 0.23703563084746843;
stInitData.ModelParameters._R[535] := 0.17433420732373484;
stInitData.ModelParameters._R[536] := 0.30180896751453995;
stInitData.ModelParameters._R[537] := 0.35455630026528762;
stInitData.ModelParameters._R[538] := 0.31470801125816983;
stInitData.ModelParameters._R[539] := 0.21812954422380954;
stInitData.ModelParameters._R[540] := 0.51051496230212812;
stInitData.ModelParameters._R[541] := 0.39317740088841913;
stInitData.ModelParameters._R[542] := 0.1633519341419945;
stInitData.ModelParameters._R[543] := 0.64727797771331863;
stInitData.ModelParameters._R[544] := 0.65285996742740715;
stInitData.ModelParameters._R[545] := 0.54553515633102234;
stInitData.ModelParameters._R[546] := 0.74054963755642045;
stInitData.ModelParameters._R[547] := 0.12547129601587542;
stInitData.ModelParameters._R[548] := 0.99638318989105135;
stInitData.ModelParameters._R[549] := 0.21449729778645679;
stInitData.ModelParameters._R[550] := 0.3732234392387892;
stInitData.ModelParameters._R[551] := 0.12840474067818322;
stInitData.ModelParameters._R[552] := 0.57289492245627871;
stInitData.ModelParameters._R[553] := 0.87767771242736869;
stInitData.ModelParameters._R[554] := 0.38660611717315441;
stInitData.ModelParameters._R[555] := 0.44028225906570007;
stInitData.ModelParameters._R[556] := 0.16433188171112439;
stInitData.ModelParameters._R[557] := 0.91205816112609328;
stInitData.ModelParameters._R[558] := 0.29411735225041125;
stInitData.ModelParameters._R[559] := 0.41005940508830607;
stInitData.ModelParameters._R[560] := 0.32859872378534849;
stInitData.ModelParameters._R[561] := 0.29233420949575506;
stInitData.ModelParameters._R[562] := 0.69168844479421454;
stInitData.ModelParameters._R[563] := 0.90362171941655101;
stInitData.ModelParameters._R[564] := 0.62573428620706872;
stInitData.ModelParameters._R[565] := 0.75556027167955442;
stInitData.ModelParameters._R[566] := 0.66320871468411313;
stInitData.ModelParameters._R[567] := 0.78111001700070637;
stInitData.ModelParameters._R[568] := 0.42646279092742245;
stInitData.ModelParameters._R[569] := 0.20350035478795181;
stInitData.ModelParameters._R[570] := 0.37105897547354949;
stInitData.ModelParameters._R[571] := 0.56248471634561814;
stInitData.ModelParameters._R[572] := 0.44129886183188138;
stInitData.ModelParameters._R[573] := 0.47816435218012121;
stInitData.ModelParameters._R[574] := 0.53768598292465752;
stInitData.ModelParameters._R[575] := 0.10746073201825783;
stInitData.ModelParameters._R[576] := 0.39443853345093394;
stInitData.ModelParameters._R[577] := 0.15581137402056405;
stInitData.ModelParameters._R[578] := 0.75790392683703178;
stInitData.ModelParameters._R[579] := 0.39428623197750301;
stInitData.ModelParameters._R[580] := 0.78824119276815563;
stInitData.ModelParameters._R[581] := 0.9634822722517935;
stInitData.ModelParameters._R[582] := 0.96730777815668423;
stInitData.ModelParameters._R[583] := 0.16348848151139422;
stInitData.ModelParameters._R[584] := 0.89633760478317093;
stInitData.ModelParameters._R[585] := 0.40960778521675345;
stInitData.ModelParameters._R[586] := 0.87338979445110976;
stInitData.ModelParameters._R[587] := 0.86737469769208975;
stInitData.ModelParameters._R[588] := 0.89389817354902978;
stInitData.ModelParameters._R[589] := 0.94037342494008702;
stInitData.ModelParameters._R[590] := 0.79070835679354423;
stInitData.ModelParameters._R[591] := 0.47491168447813348;
stInitData.ModelParameters._R[592] := 0.10881178516417116;
stInitData.ModelParameters._R[593] := 0.66452595545044868;
stInitData.ModelParameters._R[594] := 0.91904823368358557;
stInitData.ModelParameters._R[595] := 0.45734534593004617;
stInitData.ModelParameters._R[596] := 0.9678476020420651;
stInitData.ModelParameters._R[597] := 0.30464994866238704;
stInitData.ModelParameters._R[598] := 0.64768960938193298;
stInitData.ModelParameters._R[599] := 0.70719310195863161;
stInitData.ModelParameters._R[600] := 0.90708890437060574;
stInitData.ModelParameters._R[601] := 0.55366765722980282;
stInitData.ModelParameters._R[602] := 0.18427955567788756;
stInitData.ModelParameters._R[603] := 0.82088913680470621;
stInitData.ModelParameters._R[604] := 0.19652259244531506;
stInitData.ModelParameters._R[605] := 0.31492198289230178;
stInitData.ModelParameters._R[606] := 0.42452274583667504;
stInitData.ModelParameters._R[607] := 0.86790432866698519;
stInitData.ModelParameters._R[608] := 0.28882892665426618;
stInitData.ModelParameters._R[609] := 0.77688054638993043;
stInitData.ModelParameters._R[610] := 0.7580242285429607;
stInitData.ModelParameters._R[611] := 0.81401186048318386;
stInitData.ModelParameters._R[612] := 0.38521485230821573;
stInitData.ModelParameters._R[613] := 0.2175841732893537;
stInitData.ModelParameters._R[614] := 0.59401425896065496;
stInitData.ModelParameters._R[615] := 0.63413437816069063;
stInitData.ModelParameters._R[616] := 0.55814964148808532;
stInitData.ModelParameters._R[617] := 0.33803612038270159;
stInitData.ModelParameters._R[618] := 0.42252171458852761;
stInitData.ModelParameters._R[619] := 0.32441050690619977;
stInitData.ModelParameters._R[620] := 0.48271731017085817;
stInitData.ModelParameters._R[621] := 0.14321042418724406;
stInitData.ModelParameters._R[622] := 0.85423872437576942;
stInitData.ModelParameters._R[623] := 0.73560201971250772;
stInitData.ModelParameters._R[624] := 0.31389640161085108;
stInitData.ModelParameters._R[625] := 0.62905071391146072;
stInitData.ModelParameters._R[626] := 0.32016778010635571;
stInitData.ModelParameters._R[627] := 0.29559175244118951;
stInitData.ModelParameters._R[628] := 0.19044887060278048;
stInitData.ModelParameters._R[629] := 0.74149657127969126;
stInitData.ModelParameters._R[630] := 0.6735820262859441;
stInitData.ModelParameters._R[631] := 0.94970602558882855;
stInitData.ModelParameters._R[632] := 0.1666609847023835;
stInitData.ModelParameters._R[633] := 0.15857461861000366;
stInitData.ModelParameters._R[634] := 0.16248890118121506;
stInitData.ModelParameters._R[635] := 0.70648280351072346;
stInitData.ModelParameters._R[636] := 0.42373607806935443;
stInitData.ModelParameters._R[637] := 0.28219615204587345;
stInitData.ModelParameters._R[638] := 0.69963878309059879;
stInitData.ModelParameters._R[639] := 0.32199134183538636;
stInitData.ModelParameters._R[640] := 0.83878167374323609;
stInitData.ModelParameters._R[641] := 0.5190369743547768;
stInitData.ModelParameters._R[642] := 0.48013317031986757;
stInitData.ModelParameters._R[643] := 0.95004029797657041;
stInitData.ModelParameters._R[644] := 0.93639954071679399;
stInitData.ModelParameters._R[645] := 0.37119601919586154;
stInitData.ModelParameters._R[646] := 0.76199672197724377;
stInitData.ModelParameters._R[647] := 0.19979664954841675;
stInitData.ModelParameters._R[648] := 0.57122483302816307;
stInitData.ModelParameters._R[649] := 0.63998728602822152;
stInitData.ModelParameters._R[650] := 0.64935366741209588;
stInitData.ModelParameters._R[651] := 0.58254111513495888;
stInitData.ModelParameters._R[652] := 0.48177035480257635;
stInitData.ModelParameters._R[653] := 0.86483883209174295;
stInitData.ModelParameters._R[654] := 0.48483938151768591;
stInitData.ModelParameters._R[655] := 0.41817120696530763;
stInitData.ModelParameters._R[656] := 0.97826882368593127;
stInitData.ModelParameters._R[657] := 0.59792809381522538;
stInitData.ModelParameters._R[658] := 0.3890198179282981;
stInitData.ModelParameters._R[659] := 0.77097378592841459;
stInitData.ModelParameters._R[660] := 0.7496996791349243;
stInitData.ModelParameters._R[661] := 0.99777374912723993;
stInitData.ModelParameters._R[662] := 0.10290994801454834;
stInitData.ModelParameters._R[663] := 0.66030684739697132;
stInitData.ModelParameters._R[664] := 0.69767342709228319;
stInitData.ModelParameters._R[665] := 0.37248634159515359;
stInitData.ModelParameters._R[666] := 0.91880725364025184;
stInitData.ModelParameters._R[667] := 0.92632415712842942;
stInitData.ModelParameters._R[668] := 0.87116217202993251;
stInitData.ModelParameters._R[669] := 0.96349207392461111;
stInitData.ModelParameters._R[670] := 0.33562782950353776;
stInitData.ModelParameters._R[671] := 0.24476392643422418;
stInitData.ModelParameters._R[672] := 0.88244986906791956;
stInitData.ModelParameters._R[673] := 0.78382896848677119;
stInitData.ModelParameters._R[674] := 0.95312741195494033;
stInitData.ModelParameters._R[675] := 0.94891022527316438;
stInitData.ModelParameters._R[676] := 0.32296451585918662;
stInitData.ModelParameters._R[677] := 0.27542455928442083;
stInitData.ModelParameters._R[678] := 0.37822514073348712;
stInitData.ModelParameters._R[679] := 0.14715709033043103;
stInitData.ModelParameters._R[680] := 0.55426702225281343;
stInitData.ModelParameters._R[681] := 0.80915226286826314;
stInitData.ModelParameters._R[682] := 0.23940167705518919;
stInitData.ModelParameters._R[683] := 0.94881938868511984;
stInitData.ModelParameters._R[684] := 0.53391461833859599;
stInitData.ModelParameters._R[685] := 0.80728971401499128;
stInitData.ModelParameters._R[686] := 0.17653085543276839;
stInitData.ModelParameters._R[687] := 0.72481239783007467;
stInitData.ModelParameters._R[688] := 0.60745445652402474;
stInitData.ModelParameters._R[689] := 0.89473150034252968;
stInitData.ModelParameters._R[690] := 0.98710219934564536;
stInitData.ModelParameters._R[691] := 0.70053502529948808;
stInitData.ModelParameters._R[692] := 0.14542398605713416;
stInitData.ModelParameters._R[693] := 0.92202924299866873;
stInitData.ModelParameters._R[694] := 0.52331957117944827;
stInitData.ModelParameters._R[695] := 0.77659672999283624;
stInitData.ModelParameters._R[696] := 0.93280793766331449;
stInitData.ModelParameters._R[697] := 0.47128098874706914;
stInitData.ModelParameters._R[698] := 0.17764240643845475;
stInitData.ModelParameters._R[699] := 0.56994999412842307;
stInitData.ModelParameters._R[700] := 0.62677089194987867;
stInitData.ModelParameters._R[701] := 0.91350355476969991;
stInitData.ModelParameters._R[702] := 0.45303430360223373;
stInitData.ModelParameters._R[703] := 0.35819184869562282;
stInitData.ModelParameters._R[704] := 0.18736361128498802;
stInitData.ModelParameters._R[705] := 0.63183403954111217;
stInitData.ModelParameters._R[706] := 0.15579399522270077;
stInitData.ModelParameters._R[707] := 0.75846337210538184;
stInitData.ModelParameters._R[708] := 0.40834847969876709;
stInitData.ModelParameters._R[709] := 0.1404941277952248;
stInitData.ModelParameters._R[710] := 0.53124345744438195;
stInitData.ModelParameters._R[711] := 0.57099091188308604;
stInitData.ModelParameters._R[712] := 0.6273817324749259;
stInitData.ModelParameters._R[713] := 0.23138357090601497;
stInitData.ModelParameters._R[714] := 0.96247915036954257;
stInitData.ModelParameters._R[715] := 0.23009485641567534;
stInitData.ModelParameters._R[716] := 0.8044452568092173;
stInitData.ModelParameters._R[717] := 0.13633690576329752;
stInitData.ModelParameters._R[718] := 0.52373099251659672;
stInitData.ModelParameters._R[719] := 0.24969611830629895;
stInitData.ModelParameters._R[720] := 0.78756940138427101;
stInitData.ModelParameters._R[721] := 0.43468406595050835;
stInitData.ModelParameters._R[722] := 0.50632039627083891;
stInitData.ModelParameters._R[723] := 0.32419420412080768;
stInitData.ModelParameters._R[724] := 0.55681262397828646;
stInitData.ModelParameters._R[725] := 0.27306704425997719;
stInitData.ModelParameters._R[726] := 0.90030412763752554;
stInitData.ModelParameters._R[727] := 0.26661930563059327;
stInitData.ModelParameters._R[728] := 0.61136957933085279;
stInitData.ModelParameters._R[729] := 0.25099268616223624;
stInitData.ModelParameters._R[730] := 0.94819304957094208;
stInitData.ModelParameters._R[731] := 0.50360756220947267;
stInitData.ModelParameters._R[732] := 0.12466506521045945;
stInitData.ModelParameters._R[733] := 0.17734921985606711;
stInitData.ModelParameters._R[734] := 0.69622266556249202;
stInitData.ModelParameters._R[735] := 0.77277269462256093;
stInitData.ModelParameters._R[736] := 0.99630127579423977;
stInitData.ModelParameters._R[737] := 0.20534935179703351;
stInitData.ModelParameters._R[738] := 0.65580157313680043;
stInitData.ModelParameters._R[739] := 0.83806290215516954;
stInitData.ModelParameters._R[740] := 0.51439291696308609;
stInitData.ModelParameters._R[741] := 0.37417811194302419;
stInitData.ModelParameters._R[742] := 0.32433357992389422;
stInitData.ModelParameters._R[743] := 0.15849328194933748;
stInitData.ModelParameters._R[744] := 0.67596845780323034;
stInitData.ModelParameters._R[745] := 0.84049817943596983;
stInitData.ModelParameters._R[746] := 0.99425722778597025;
stInitData.ModelParameters._R[747] := 0.27833336878156489;
stInitData.ModelParameters._R[748] := 0.7936361408990571;
stInitData.ModelParameters._R[749] := 0.38987732947360543;
stInitData.ModelParameters._R[750] := 0.13636941755589962;
stInitData.ModelParameters._R[751] := 0.44176134686839463;
stInitData.ModelParameters._R[752] := 0.73344734730813732;
stInitData.ModelParameters._R[753] := 0.57320193242772932;
stInitData.ModelParameters._R[754] := 0.38362107708531834;
stInitData.ModelParameters._R[755] := 0.59876238101381341;
stInitData.ModelParameters._R[756] := 0.23053021146955438;
stInitData.ModelParameters._R[757] := 0.59182147000380925;
stInitData.ModelParameters._R[758] := 0.59254382446743648;
stInitData.ModelParameters._R[759] := 0.21191430409611717;
stInitData.ModelParameters._R[760] := 0.43602342473099942;
stInitData.ModelParameters._R[761] := 0.68663004478297973;
stInitData.ModelParameters._R[762] := 0.1086330751280379;
stInitData.ModelParameters._R[763] := 0.19364861429499597;
stInitData.ModelParameters._R[764] := 0.77993998468245962;
stInitData.ModelParameters._R[765] := 0.59328569133520404;
stInitData.ModelParameters._R[766] := 0.90103559505145203;
stInitData.ModelParameters._R[767] := 0.35842579441827482;
stInitData.ModelParameters._R[768] := 0.55769055117904576;
stInitData.ModelParameters._R[769] := 0.79043334900404272;
stInitData.ModelParameters._R[770] := 0.54027481226663987;
stInitData.ModelParameters._R[771] := 0.75735151161551739;
stInitData.ModelParameters._R[772] := 0.52320829671041424;
stInitData.ModelParameters._R[773] := 0.81085107336719042;
stInitData.ModelParameters._R[774] := 0.79087348702003646;
stInitData.ModelParameters._R[775] := 0.46089733562703583;
stInitData.ModelParameters._R[776] := 0.44698932250638679;
stInitData.ModelParameters._R[777] := 0.20433845415768337;
stInitData.ModelParameters._R[778] := 0.12696709219509666;
stInitData.ModelParameters._R[779] := 0.41395467590738433;
stInitData.ModelParameters._R[780] := 0.29537437407896677;
stInitData.ModelParameters._R[781] := 0.84684132647456001;
stInitData.ModelParameters._R[782] := 0.41931731530476524;
stInitData.ModelParameters._R[783] := 0.58352406000793799;
stInitData.ModelParameters._R[784] := 0.82454072929927946;
stInitData.ModelParameters._R[785] := 0.63476221432814373;
stInitData.ModelParameters._R[786] := 0.91610082071571231;
stInitData.ModelParameters._R[787] := 0.70874315740251381;
stInitData.ModelParameters._R[788] := 0.27190384356577263;
stInitData.ModelParameters._R[789] := 0.98080986159300854;
stInitData.ModelParameters._R[790] := 0.68307809679649178;
stInitData.ModelParameters._R[791] := 0.80732150082971976;
stInitData.ModelParameters._R[792] := 0.46083257317841164;
stInitData.ModelParameters._R[793] := 0.33654764706212337;
stInitData.ModelParameters._R[794] := 0.38387197118902994;
stInitData.ModelParameters._R[795] := 0.53456972414138237;
stInitData.ModelParameters._R[796] := 0.25736293189789672;
stInitData.ModelParameters._R[797] := 0.6636663212117565;
stInitData.ModelParameters._R[798] := 0.74782083423276213;
stInitData.ModelParameters._R[799] := 0.28532393031724068;
stInitData.ModelParameters._R[800] := 0.66861657161269095;
stInitData.ModelParameters._R[801] := 0.72619310210189281;
stInitData.ModelParameters._R[802] := 0.18960560318724656;
stInitData.ModelParameters._R[803] := 0.13370052187830483;
stInitData.ModelParameters._R[804] := 0.92603678881215268;
stInitData.ModelParameters._R[805] := 0.48271054930388746;
stInitData.ModelParameters._R[806] := 0.90201923810745843;
stInitData.ModelParameters._R[807] := 0.50767454762912823;
stInitData.ModelParameters._R[808] := 0.31525464212822774;
stInitData.ModelParameters._R[809] := 0.6585616956161322;
stInitData.ModelParameters._R[810] := 0.8660674749426942;
stInitData.ModelParameters._R[811] := 0.86646320639452201;
stInitData.ModelParameters._R[812] := 0.74694550271219906;
stInitData.ModelParameters._R[813] := 0.33528237308901199;
stInitData.ModelParameters._R[814] := 0.64513130871540636;
stInitData.ModelParameters._R[815] := 0.31769600797512521;
stInitData.ModelParameters._R[816] := 0.74516996526665047;
stInitData.ModelParameters._R[817] := 0.58422686412877112;
stInitData.ModelParameters._R[818] := 0.140738485272002;
stInitData.ModelParameters._R[819] := 0.39416231556255132;
stInitData.ModelParameters._R[820] := 0.57447260888789198;
stInitData.ModelParameters._R[821] := 0.64680144476606971;
stInitData.ModelParameters._R[822] := 0.4425588358261473;
stInitData.ModelParameters._R[823] := 0.27962997513483423;
stInitData.ModelParameters._R[824] := 0.938832045064522;
stInitData.ModelParameters._R[825] := 0.86397369072126062;
stInitData.ModelParameters._R[826] := 0.56902805366922626;
stInitData.ModelParameters._R[827] := 0.26703044907905571;
stInitData.ModelParameters._R[828] := 0.14554832611760488;
stInitData.ModelParameters._R[829] := 0.96868586742315532;
stInitData.ModelParameters._R[830] := 0.60189478255512618;
stInitData.ModelParameters._R[831] := 0.82373799642592205;
stInitData.ModelParameters._R[832] := 0.32546272655028519;
stInitData.ModelParameters._R[833] := 0.40513767095809117;
stInitData.ModelParameters._R[834] := 0.74334503837402399;
stInitData.ModelParameters._R[835] := 0.41377599240629759;
stInitData.ModelParameters._R[836] := 0.12605420078542331;
stInitData.ModelParameters._R[837] := 0.59149857260650018;
stInitData.ModelParameters._R[838] := 0.26020903659320088;
stInitData.ModelParameters._R[839] := 0.81356452088076248;
stInitData.ModelParameters._R[840] := 0.55760877718928947;
stInitData.ModelParameters._R[841] := 0.32329858451012466;
stInitData.ModelParameters._R[842] := 0.71528321302749376;
stInitData.ModelParameters._R[843] := 0.5369967100100973;
stInitData.ModelParameters._R[844] := 0.59716509769537707;
stInitData.ModelParameters._R[845] := 0.69725833302161455;
stInitData.ModelParameters._R[846] := 0.5365341112031724;
stInitData.ModelParameters._R[847] := 0.27574002962958782;
stInitData.ModelParameters._R[848] := 0.61863189431428112;
stInitData.ModelParameters._R[849] := 0.63849478851732056;
stInitData.ModelParameters._R[850] := 0.23001735226740999;
stInitData.ModelParameters._R[851] := 0.14350767293586159;
stInitData.ModelParameters._R[852] := 0.16587153349680883;
stInitData.ModelParameters._R[853] := 0.63965021490394525;
stInitData.ModelParameters._R[854] := 0.51871967989704992;
stInitData.ModelParameters._R[855] := 0.60397265800126654;
stInitData.ModelParameters._R[856] := 0.87460730638746964;
stInitData.ModelParameters._R[857] := 0.24387498091187673;
stInitData.ModelParameters._R[858] := 0.13139419594356672;
stInitData.ModelParameters._R[859] := 0.41249817684816903;
stInitData.ModelParameters._R[860] := 0.76727759143920438;
stInitData.ModelParameters._R[861] := 0.18110971770706127;
stInitData.ModelParameters._R[862] := 0.24211594736805578;
stInitData.ModelParameters._R[863] := 0.73406980183760007;
stInitData.ModelParameters._R[864] := 0.62457319284072144;
stInitData.ModelParameters._R[865] := 0.24484785793347486;
stInitData.ModelParameters._R[866] := 0.35842114393228808;
stInitData.ModelParameters._R[867] := 0.24760120422385049;
stInitData.ModelParameters._R[868] := 0.49477766373818355;
stInitData.ModelParameters._R[869] := 0.9751764840703967;
stInitData.ModelParameters._R[870] := 0.34232309087644164;
stInitData.ModelParameters._R[871] := 0.84120297706595992;
stInitData.ModelParameters._R[872] := 0.75270855031771888;
stInitData.ModelParameters._R[873] := 0.93102059845208507;
stInitData.ModelParameters._R[874] := 0.22683378226263864;
stInitData.ModelParameters._R[875] := 0.9529578085156013;
stInitData.ModelParameters._R[876] := 0.43078713619059184;
stInitData.ModelParameters._R[877] := 0.72589742344817354;
stInitData.ModelParameters._R[878] := 0.40896084454863424;
stInitData.ModelParameters._R[879] := 0.20128140673286465;
stInitData.ModelParameters._R[880] := 0.11677176587322879;
stInitData.ModelParameters._R[881] := 0.46363876464717901;
stInitData.ModelParameters._R[882] := 0.23879942268749535;
stInitData.ModelParameters._R[883] := 0.5999014645121763;
stInitData.ModelParameters._R[884] := 0.99452529184847349;
stInitData.ModelParameters._R[885] := 0.70565840186805695;
stInitData.ModelParameters._R[886] := 0.23177209952452549;
stInitData.ModelParameters._R[887] := 0.54268424012228245;
stInitData.ModelParameters._R[888] := 0.42130869513364333;
stInitData.ModelParameters._R[889] := 0.47771947719440255;
stInitData.ModelParameters._R[890] := 0.52571303743103248;
stInitData.ModelParameters._R[891] := 0.90410652581366646;
stInitData.ModelParameters._R[892] := 0.43106833714437687;
stInitData.ModelParameters._R[893] := 0.80085479804277415;
stInitData.ModelParameters._R[894] := 0.19179825609965817;
stInitData.ModelParameters._R[895] := 0.46438276218677088;
stInitData.ModelParameters._R[896] := 0.5972722144894359;
stInitData.ModelParameters._R[897] := 0.22227704279892171;
stInitData.ModelParameters._R[898] := 0.85244401000086134;
stInitData.ModelParameters._R[899] := 0.33819987813289565;
stInitData.ModelParameters._R[900] := 0.93468798155282484;
stInitData.ModelParameters._R[901] := 0.24912584307195967;
stInitData.ModelParameters._R[902] := 0.79588153946353346;
stInitData.ModelParameters._R[903] := 0.6916772425660237;
stInitData.ModelParameters._R[904] := 0.6990512834667616;
stInitData.ModelParameters._R[905] := 0.2637693226847283;
stInitData.ModelParameters._R[906] := 0.88109903959431035;
stInitData.ModelParameters._R[907] := 0.79512158296108215;
stInitData.ModelParameters._R[908] := 0.89224849085687674;
stInitData.ModelParameters._R[909] := 0.4474035030089103;
stInitData.ModelParameters._R[910] := 0.54496990097287323;
stInitData.ModelParameters._R[911] := 0.30243324277608918;
stInitData.ModelParameters._R[912] := 0.31982074694532103;
stInitData.ModelParameters._R[913] := 0.8362838281016638;
stInitData.ModelParameters._R[914] := 0.86207203136320232;
stInitData.ModelParameters._R[915] := 0.82755126452388139;
stInitData.ModelParameters._R[916] := 0.1539158514870278;
stInitData.ModelParameters._R[917] := 0.14358305830231843;
stInitData.ModelParameters._R[918] := 0.65382559893814296;
stInitData.ModelParameters._R[919] := 0.61988660109951377;
stInitData.ModelParameters._R[920] := 0.43494973899581024;
stInitData.ModelParameters._R[921] := 0.92235279691003558;
stInitData.ModelParameters._R[922] := 0.26214432791526615;
stInitData.ModelParameters._R[923] := 0.47794362366033849;
stInitData.ModelParameters._R[924] := 0.26228891987733666;
stInitData.ModelParameters._R[925] := 0.65281887323430932;
stInitData.ModelParameters._R[926] := 0.49254960407085624;
stInitData.ModelParameters._R[927] := 0.44435119672081913;
stInitData.ModelParameters._R[928] := 0.80252073646956068;
stInitData.ModelParameters._R[929] := 0.82366623852454401;
stInitData.ModelParameters._R[930] := 0.23167544340457819;
stInitData.ModelParameters._R[931] := 0.56670530712588241;
stInitData.ModelParameters._R[932] := 0.10473672025966008;
stInitData.ModelParameters._R[933] := 0.72275760871988415;
stInitData.ModelParameters._R[934] := 0.17553402687878894;
stInitData.ModelParameters._R[935] := 0.5722526525571876;
stInitData.ModelParameters._R[936] := 0.67628475217127149;
stInitData.ModelParameters._R[937] := 0.18112931816317593;
stInitData.ModelParameters._R[938] := 0.73379350162183909;
stInitData.ModelParameters._R[939] := 0.98587356826343653;
stInitData.ModelParameters._R[940] := 0.93952244910100802;
stInitData.ModelParameters._R[941] := 0.29922460448221566;
stInitData.ModelParameters._R[942] := 0.5795783704530556;
stInitData.ModelParameters._R[943] := 0.84598858527212706;
stInitData.ModelParameters._R[944] := 0.2898228584300343;
stInitData.ModelParameters._R[945] := 0.42638847278753944;
stInitData.ModelParameters._R[946] := 0.39763003089449778;
stInitData.ModelParameters._R[947] := 0.50357444751200664;
stInitData.ModelParameters._R[948] := 0.45875460040775273;
stInitData.ModelParameters._R[949] := 0.66680613051452908;
stInitData.ModelParameters._R[950] := 0.18842772992692627;
stInitData.ModelParameters._R[951] := 0.62242742136622486;
stInitData.ModelParameters._R[952] := 0.71134936145340577;
stInitData.ModelParameters._R[953] := 0.61804150248160572;
stInitData.ModelParameters._R[954] := 0.94150916117867345;
stInitData.ModelParameters._R[955] := 0.52857853058889415;
stInitData.ModelParameters._R[956] := 0.87649671642230664;
stInitData.ModelParameters._R[957] := 0.61310925188171872;
stInitData.ModelParameters._R[958] := 0.43953858948383506;
stInitData.ModelParameters._R[959] := 0.15507808778586601;
stInitData.ModelParameters._R[960] := 0.82167916141602571;
stInitData.ModelParameters._R[961] := 0.84718431491508173;
stInitData.ModelParameters._R[962] := 0.63357566636407159;
stInitData.ModelParameters._R[963] := 0.63328057584162212;
stInitData.ModelParameters._R[964] := 0.21613986113153125;
stInitData.ModelParameters._R[965] := 0.84963628586623385;
stInitData.ModelParameters._R[966] := 0.14147919918408008;
stInitData.ModelParameters._R[967] := 0.34141258837206856;
stInitData.ModelParameters._R[968] := 0.80356986036995848;
stInitData.ModelParameters._R[969] := 0.83905761570014348;
stInitData.ModelParameters._R[970] := 0.55706515845815319;
stInitData.ModelParameters._R[971] := 0.4538582813447033;
stInitData.ModelParameters._R[972] := 0.94498159714127483;
stInitData.ModelParameters._R[973] := 0.28414030006425572;
stInitData.ModelParameters._R[974] := 0.2709214092147787;
stInitData.ModelParameters._R[975] := 0.90453253544418155;
stInitData.ModelParameters._R[976] := 0.43920604326235868;
stInitData.ModelParameters._R[977] := 0.87817716632381027;
stInitData.ModelParameters._R[978] := 0.15331720151876785;
stInitData.ModelParameters._R[979] := 0.84002397281270513;
stInitData.ModelParameters._R[980] := 0.54166231761190498;
stInitData.ModelParameters._R[981] := 0.31755877977612601;
stInitData.ModelParameters._R[982] := 0.45814137624691542;
stInitData.ModelParameters._R[983] := 0.39603272904198339;
stInitData.ModelParameters._R[984] := 0.20900501603606386;
stInitData.ModelParameters._R[985] := 0.19170405906809668;
stInitData.ModelParameters._R[986] := 0.78681433359954389;
stInitData.ModelParameters._R[987] := 0.71481207634625488;
stInitData.ModelParameters._R[988] := 0.94096083001728581;
stInitData.ModelParameters._R[989] := 0.15250608787471198;
stInitData.ModelParameters._R[990] := 0.68978082940189334;
stInitData.ModelParameters._R[991] := 0.16087658083046907;
stInitData.ModelParameters._R[992] := 0.12164603469164069;
stInitData.ModelParameters._R[993] := 0.36823941528984128;
stInitData.ModelParameters._R[994] := 0.78961413186953955;
stInitData.ModelParameters._R[995] := 0.25383178475075019;
stInitData.ModelParameters._R[996] := 0.92483318769842582;
stInitData.ModelParameters._R[997] := 0.41346397022867099;
stInitData.ModelParameters._R[998] := 0.40866122739504918;
stInitData.ModelParameters._R[999] := 0.5313017095839534;
stInitData.ModelParameters._R[1000] := 0.33431185552925557;
stInitData.ModelParameters._R[1001] := 0.46690248408804702;
stInitData.ModelParameters._R[1002] := 0.77830199182800874;
stInitData.ModelParameters._R[1003] := 0.54471677774186533;
stInitData.ModelParameters._R[1004] := 0.43086685277857095;
stInitData.ModelParameters._R[1005] := 0.21475840052213768;
stInitData.ModelParameters._R[1006] := 0.7885650963132893;
stInitData.ModelParameters._R[1007] := 0.39862473124918651;
stInitData.ModelParameters._R[1008] := 0.23931437783161141;
stInitData.ModelParameters._R[1009] := 0.82144926818172392;
stInitData.ModelParameters._R[1010] := 0.71606512599479044;
stInitData.ModelParameters._R[1011] := 0.2681834913538097;
stInitData.ModelParameters._R[1012] := 0.72275721013731598;
stInitData.ModelParameters._R[1013] := 0.29856174508042066;
stInitData.ModelParameters._R[1014] := 0.82096134688275135;
stInitData.ModelParameters._R[1015] := 0.24601582863622348;
stInitData.ModelParameters._R[1016] := 0.78262773139402231;
stInitData.ModelParameters._R[1017] := 0.14777025139083497;
stInitData.ModelParameters._R[1018] := 0.54537331514670395;
stInitData.ModelParameters._R[1019] := 0.14443340640613159;
stInitData.ModelParameters._R[1020] := 0.54741286040993342;
stInitData.ModelParameters._R[1021] := 0.71209452624165948;
stInitData.ModelParameters._R[1022] := 0.2605984093346882;
stInitData.ModelParameters._R[1023] := 0.68717054178181092;
stInitData.ModelParameters._R[1024] := 0.1773898236165164;
stInitData.ModelParameters._R[1025] := 0.29718641487061259;
stInitData.ModelParameters._R[1026] := 0.21885939935224186;
stInitData.ModelParameters._R[1027] := 0.25819864885781707;
stInitData.ModelParameters._R[1028] := 0.3700205617935477;
stInitData.ModelParameters._R[1029] := 0.13911798176489926;
stInitData.ModelParameters._R[1030] := 0.9435575093063181;
stInitData.ModelParameters._R[1031] := 0.14768166376480335;
stInitData.ModelParameters._R[1032] := 0.3946596722082848;
stInitData.ModelParameters._R[1033] := 0.39032604007696736;
stInitData.ModelParameters._R[1034] := 0.71362093519298631;
stInitData.ModelParameters._R[1035] := 0.44077219989795513;
stInitData.ModelParameters._R[1036] := 0.71641575999652785;
stInitData.ModelParameters._R[1037] := 0.61337572670030793;
stInitData.ModelParameters._R[1038] := 0.62242419522520254;
stInitData.ModelParameters._R[1039] := 0.28489862565676377;
stInitData.ModelParameters._R[1040] := 0.83053860169061433;
stInitData.ModelParameters._R[1041] := 0.61304387021442386;
stInitData.ModelParameters._R[1042] := 0.96524024371655059;
stInitData.ModelParameters._R[1043] := 0.97755460854447196;
stInitData.ModelParameters._R[1044] := 0.71578373734559797;
stInitData.ModelParameters._R[1045] := 0.40778897679256798;
stInitData.ModelParameters._R[1046] := 0.30573393497027113;
stInitData.ModelParameters._R[1047] := 0.95887422332328187;
stInitData.ModelParameters._R[1048] := 0.25193305786467479;
stInitData.ModelParameters._R[1049] := 0.390631812713511;
stInitData.ModelParameters._R[1050] := 0.46783753340069256;
stInitData.ModelParameters._R[1051] := 0.96612377744826805;
stInitData.ModelParameters._R[1052] := 0.63091958493609657;
stInitData.ModelParameters._R[1053] := 0.63016378170703236;
stInitData.ModelParameters._R[1054] := 0.18048324633768714;
stInitData.ModelParameters._R[1055] := 0.37452023792420375;
stInitData.ModelParameters._R[1056] := 0.32489167674679942;
stInitData.ModelParameters._R[1057] := 0.65194596968070717;
stInitData.ModelParameters._R[1058] := 0.96658971627533907;
stInitData.ModelParameters._R[1059] := 0.91230727427175584;
stInitData.ModelParameters._R[1060] := 0.12581983213445683;
stInitData.ModelParameters._R[1061] := 0.88662545451451813;
stInitData.ModelParameters._R[1062] := 0.361797764378192;
stInitData.ModelParameters._R[1063] := 0.83529547583694486;
stInitData.ModelParameters._R[1064] := 0.58324739550919691;
stInitData.ModelParameters._R[1065] := 0.80725023544827579;
stInitData.ModelParameters._R[1066] := 0.79925417406727717;
stInitData.ModelParameters._R[1067] := 0.7887249957959499;
stInitData.ModelParameters._R[1068] := 0.70206332391042059;
stInitData.ModelParameters._R[1069] := 0.11235019859950163;
stInitData.ModelParameters._R[1070] := 0.29530254419420071;
stInitData.ModelParameters._R[1071] := 0.52013417934187611;
stInitData.ModelParameters._R[1072] := 0.28649652648113288;
stInitData.ModelParameters._R[1073] := 0.3702707829157611;
stInitData.ModelParameters._R[1074] := 0.13774056198364787;
stInitData.ModelParameters._R[1075] := 0.19750257295660933;
stInitData.ModelParameters._R[1076] := 0.21442309054350861;
stInitData.ModelParameters._R[1077] := 0.90631807755888594;
stInitData.ModelParameters._R[1078] := 0.31887395620636616;
stInitData.ModelParameters._R[1079] := 0.63856039183546176;
stInitData.ModelParameters._R[1080] := 0.61457722478170163;
stInitData.ModelParameters._R[1081] := 0.87058977437660545;
stInitData.ModelParameters._R[1082] := 0.50197286280161946;
stInitData.ModelParameters._R[1083] := 0.11826103813696881;
stInitData.ModelParameters._R[1084] := 0.96086693875008877;
stInitData.ModelParameters._R[1085] := 0.88885829612465883;
stInitData.ModelParameters._R[1086] := 0.4884068888355303;
stInitData.ModelParameters._R[1087] := 0.54875971596269624;
stInitData.ModelParameters._R[1088] := 0.36532285318353108;
stInitData.ModelParameters._R[1089] := 0.9667632246001332;
stInitData.ModelParameters._R[1090] := 0.99264305539426712;
stInitData.ModelParameters._R[1091] := 0.7177505161813531;
stInitData.ModelParameters._R[1092] := 0.77089286090563414;
stInitData.ModelParameters._R[1093] := 0.75405048265506291;
stInitData.ModelParameters._R[1094] := 0.98508353348242428;
stInitData.ModelParameters._R[1095] := 0.92064127311288058;
stInitData.ModelParameters._R[1096] := 0.80448666120281187;
stInitData.ModelParameters._R[1097] := 0.44199588970892345;
stInitData.ModelParameters._R[1098] := 0.40822740113402245;
stInitData.ModelParameters._R[1099] := 0.49589959445911758;
stInitData.ModelParameters._R[1100] := 0.45722761344379248;
stInitData.ModelParameters._R[1101] := 0.38120116465914944;
stInitData.ModelParameters._R[1102] := 0.18633158332492389;
stInitData.ModelParameters._R[1103] := 0.92540734514952083;
stInitData.ModelParameters._R[1104] := 0.9035957745281602;
stInitData.ModelParameters._R[1105] := 0.26354361377249341;
stInitData.ModelParameters._R[1106] := 0.60013698527925785;
stInitData.ModelParameters._R[1107] := 0.57954126020944197;
stInitData.ModelParameters._R[1108] := 0.88628669787099879;
stInitData.ModelParameters._R[1109] := 0.75639489776739266;
stInitData.ModelParameters._R[1110] := 0.17243115712791579;
stInitData.ModelParameters._R[1111] := 0.66611207405674788;
stInitData.ModelParameters._R[1112] := 0.49702785365350732;
stInitData.ModelParameters._R[1113] := 0.25259001440680451;
stInitData.ModelParameters._R[1114] := 0.66887658700514974;
stInitData.ModelParameters._R[1115] := 0.13045324996832172;
stInitData.ModelParameters._R[1116] := 0.9164098143900179;
stInitData.ModelParameters._R[1117] := 0.11316599462856483;
stInitData.ModelParameters._R[1118] := 0.73705484619552097;
stInitData.ModelParameters._R[1119] := 0.58623674635438228;
stInitData.ModelParameters._R[1120] := 0.73313710051085612;
stInitData.ModelParameters._R[1121] := 0.78265883953759252;
stInitData.ModelParameters._R[1122] := 0.48163428242175566;
stInitData.ModelParameters._R[1123] := 0.92693565921213505;
stInitData.ModelParameters._R[1124] := 0.12326128273393448;
stInitData.ModelParameters._R[1125] := 0.50509560311703627;
stInitData.ModelParameters._R[1126] := 0.23115032401103799;
stInitData.ModelParameters._R[1127] := 0.98652790141051605;
stInitData.ModelParameters._R[1128] := 0.89481014011228899;
stInitData.ModelParameters._R[1129] := 0.5291129323764665;
stInitData.ModelParameters._R[1130] := 0.5398321860403692;
stInitData.ModelParameters._R[1131] := 0.84412685233753737;
stInitData.ModelParameters._R[1132] := 0.20854448240140178;
stInitData.ModelParameters._R[1133] := 0.71270583272140664;
stInitData.ModelParameters._R[1134] := 0.62361929218720902;
stInitData.ModelParameters._R[1135] := 0.24710195192164988;
stInitData.ModelParameters._R[1136] := 0.22069333590830109;
stInitData.ModelParameters._R[1137] := 0.2726117268703761;
stInitData.ModelParameters._R[1138] := 0.64335203606313829;
stInitData.ModelParameters._R[1139] := 0.85834839070993618;
stInitData.ModelParameters._R[1140] := 0.65088990894232213;
stInitData.ModelParameters._R[1141] := 0.81894529292966101;
stInitData.ModelParameters._R[1142] := 0.16161458068427084;
stInitData.ModelParameters._R[1143] := 0.68448937798039799;
stInitData.ModelParameters._R[1144] := 0.53757886314057379;
stInitData.ModelParameters._R[1145] := 0.32216492746294023;
stInitData.ModelParameters._R[1146] := 0.76530470144296692;
stInitData.ModelParameters._R[1147] := 0.40427504770441569;
stInitData.ModelParameters._R[1148] := 0.66798234573807214;
stInitData.ModelParameters._R[1149] := 0.41329560862627257;
stInitData.ModelParameters._R[1150] := 0.39475802088441436;
stInitData.ModelParameters._R[1151] := 0.5200188864935138;
stInitData.ModelParameters._R[1152] := 0.45306267276868784;
stInitData.ModelParameters._R[1153] := 0.50036208003972571;
stInitData.ModelParameters._R[1154] := 0.38059696453574854;
stInitData.ModelParameters._R[1155] := 0.20950555513620678;
stInitData.ModelParameters._R[1156] := 0.2948131896534949;
stInitData.ModelParameters._R[1157] := 0.49383551622577737;
stInitData.ModelParameters._R[1158] := 0.56501846297150382;
stInitData.ModelParameters._R[1159] := 0.87026252224667844;
stInitData.ModelParameters._R[1160] := 0.52921744887265643;
stInitData.ModelParameters._R[1161] := 0.74659217236599995;
stInitData.ModelParameters._R[1162] := 0.13061245164843696;
stInitData.ModelParameters._R[1163] := 0.65825631937204343;
stInitData.ModelParameters._R[1164] := 0.90677396278377542;
stInitData.ModelParameters._R[1165] := 0.45518542309830801;
stInitData.ModelParameters._R[1166] := 0.30018154237521683;
stInitData.ModelParameters._R[1167] := 0.41554919996019768;
stInitData.ModelParameters._R[1168] := 0.48353598887606497;
stInitData.ModelParameters._R[1169] := 0.29123992747521549;
stInitData.ModelParameters._R[1170] := 0.38386251836424023;
stInitData.ModelParameters._R[1171] := 0.99630087279062784;
stInitData.ModelParameters._R[1172] := 0.53777258053345045;
stInitData.ModelParameters._R[1173] := 0.26743068727600883;
stInitData.ModelParameters._R[1174] := 0.10049631084793215;
stInitData.ModelParameters._R[1175] := 0.94525412121404262;
stInitData.ModelParameters._R[1176] := 0.55340084878497009;
stInitData.ModelParameters._R[1177] := 0.73001650319513245;
stInitData.ModelParameters._R[1178] := 0.94007234851136623;
stInitData.ModelParameters._R[1179] := 0.35321770149114884;
stInitData.ModelParameters._R[1180] := 0.42895935705459098;
stInitData.ModelParameters._R[1181] := 0.98550920047059887;
stInitData.ModelParameters._R[1182] := 0.10867590805271171;
stInitData.ModelParameters._R[1183] := 0.90124133522403727;
stInitData.ModelParameters._R[1184] := 0.60438452769874318;
stInitData.ModelParameters._R[1185] := 0.44853307875675119;
stInitData.ModelParameters._R[1186] := 0.63134280153951128;
stInitData.ModelParameters._R[1187] := 0.70557890699435721;
stInitData.ModelParameters._R[1188] := 0.62982764462573959;
stInitData.ModelParameters._R[1189] := 0.65067932223273961;
stInitData.ModelParameters._R[1190] := 0.70920860089898718;
stInitData.ModelParameters._R[1191] := 0.98324564389228108;
stInitData.ModelParameters._R[1192] := 0.20418271675782845;
stInitData.ModelParameters._R[1193] := 0.74972048323491758;
stInitData.ModelParameters._R[1194] := 0.53177583627777936;
stInitData.ModelParameters._R[1195] := 0.53572395402402684;
stInitData.ModelParameters._R[1196] := 0.61914658916336829;
stInitData.ModelParameters._R[1197] := 0.56342618476388195;
stInitData.ModelParameters._R[1198] := 0.15808622335323924;
stInitData.ModelParameters._R[1199] := 0.92367198527541616;
stInitData.ModelParameters._R[1200] := 0.42498891556857543;
stInitData.ModelParameters._R[1201] := 0.28247007821979242;
stInitData.ModelParameters._R[1202] := 0.45002718523375118;
stInitData.ModelParameters._R[1203] := 0.97735824967581286;
stInitData.ModelParameters._R[1204] := 0.7468420562402569;
stInitData.ModelParameters._R[1205] := 0.25160760713316543;
stInitData.ModelParameters._R[1206] := 0.94172687573745617;
stInitData.ModelParameters._R[1207] := 0.1061998481422346;
stInitData.ModelParameters._R[1208] := 0.58003320857831286;
stInitData.ModelParameters._R[1209] := 0.74704407250584326;
stInitData.ModelParameters._R[1210] := 0.57757096767110327;
stInitData.ModelParameters._R[1211] := 0.43435103717418111;
stInitData.ModelParameters._R[1212] := 0.2020793180101178;
stInitData.ModelParameters._R[1213] := 0.62627247608057612;
stInitData.ModelParameters._R[1214] := 0.82186251889342499;
stInitData.ModelParameters._R[1215] := 0.53095120011112173;
stInitData.ModelParameters._R[1216] := 0.37184649565457129;
stInitData.ModelParameters._R[1217] := 0.34030094109941611;
stInitData.ModelParameters._R[1218] := 0.59725842871830914;
stInitData.ModelParameters._R[1219] := 0.94681122391259598;
stInitData.ModelParameters._R[1220] := 0.83710312241253915;
stInitData.ModelParameters._R[1221] := 0.67622410312433534;
stInitData.ModelParameters._R[1222] := 0.88753562462261615;
stInitData.ModelParameters._R[1223] := 0.51879853206467141;
stInitData.ModelParameters._R[1224] := 0.68961564745090509;
stInitData.ModelParameters._R[1225] := 0.46175730932583403;
stInitData.ModelParameters._R[1226] := 0.94797601307869162;
stInitData.ModelParameters._R[1227] := 0.72372821844459279;
stInitData.ModelParameters._R[1228] := 0.16438726969795953;
stInitData.ModelParameters._R[1229] := 0.13835974147128757;
stInitData.ModelParameters._R[1230] := 0.12943119382160523;
stInitData.ModelParameters._R[1231] := 0.4772036642376335;
stInitData.ModelParameters._R[1232] := 0.85243588327884878;
stInitData.ModelParameters._R[1233] := 0.78749993311003352;
stInitData.ModelParameters._R[1234] := 0.4528465601156989;
stInitData.ModelParameters._R[1235] := 0.87893815653149421;
stInitData.ModelParameters._R[1236] := 0.27964906357751063;
stInitData.ModelParameters._R[1237] := 0.33342303863161582;
stInitData.ModelParameters._R[1238] := 0.15389321863429692;
stInitData.ModelParameters._R[1239] := 0.180192686564426;
stInitData.ModelParameters._R[1240] := 0.19700351536540595;
stInitData.ModelParameters._R[1241] := 0.70579682717636505;
stInitData.ModelParameters._R[1242] := 0.13596038931173024;
stInitData.ModelParameters._R[1243] := 0.97907458775375356;
stInitData.ModelParameters._R[1244] := 0.19738855834715624;
stInitData.ModelParameters._R[1245] := 0.10513913207624075;
stInitData.ModelParameters._R[1246] := 0.29652881788159768;
stInitData.ModelParameters._R[1247] := 0.35272107513901052;
stInitData.ModelParameters._R[1248] := 0.90963885819303614;
stInitData.ModelParameters._R[1249] := 0.76527467886203648;
stInitData.ModelParameters._R[1250] := 0.52951025065035073;
stInitData.ModelParameters._R[1251] := 0.3906673856962154;
stInitData.ModelParameters._R[1252] := 0.73581466670551188;
stInitData.ModelParameters._R[1253] := 0.96560976676790533;
stInitData.ModelParameters._R[1254] := 0.7113475714837908;
stInitData.ModelParameters._R[1255] := 0.96875755731210966;
stInitData.ModelParameters._R[1256] := 0.19586865555828592;
stInitData.ModelParameters._R[1257] := 0.84843938838708299;
stInitData.ModelParameters._R[1258] := 0.77922690820204876;
stInitData.ModelParameters._R[1259] := 0.68341130763312552;
stInitData.ModelParameters._R[1260] := 0.28203563159861611;
stInitData.ModelParameters._R[1261] := 0.71284649206907569;
stInitData.ModelParameters._R[1262] := 0.28662672796160404;
stInitData.ModelParameters._R[1263] := 0.3272987574213917;
stInitData.ModelParameters._R[1264] := 0.34476678902899738;
stInitData.ModelParameters._R[1265] := 0.12254088780220254;
stInitData.ModelParameters._R[1266] := 0.29620483823047206;
stInitData.ModelParameters._R[1267] := 0.17399466196220958;
stInitData.ModelParameters._R[1268] := 0.42691086226314201;
stInitData.ModelParameters._R[1269] := 0.25272367772322724;
stInitData.ModelParameters._R[1270] := 0.91599775646513681;
stInitData.ModelParameters._R[1271] := 0.90411280462433841;
stInitData.ModelParameters._R[1272] := 0.56865406186694856;
stInitData.ModelParameters._R[1273] := 0.22248701202952786;
stInitData.ModelParameters._R[1274] := 0.62224495062011453;
stInitData.ModelParameters._R[1275] := 0.52126798974472943;
stInitData.ModelParameters._R[1276] := 0.38450867171970948;
stInitData.ModelParameters._R[1277] := 0.51924647381074118;
stInitData.ModelParameters._R[1278] := 0.55725579813340498;
stInitData.ModelParameters._R[1279] := 0.99833544004540065;
stInitData.ModelParameters._R[1280] := 0.50972708104615672;
stInitData.ModelParameters._R[1281] := 0.75897828495633524;
stInitData.ModelParameters._R[1282] := 0.28758607830977434;
stInitData.ModelParameters._R[1283] := 0.98068272282459157;
stInitData.ModelParameters._R[1284] := 0.10776798154658644;
stInitData.ModelParameters._R[1285] := 0.28003011635376629;
stInitData.ModelParameters._R[1286] := 0.573008103759856;
stInitData.ModelParameters._R[1287] := 0.55281889573341347;
stInitData.ModelParameters._R[1288] := 0.45186870178506289;
stInitData.ModelParameters._R[1289] := 0.54666225774555355;
stInitData.ModelParameters._R[1290] := 0.72214256444267289;
stInitData.ModelParameters._R[1291] := 0.83257934218519269;
stInitData.ModelParameters._R[1292] := 0.38573681323568798;
stInitData.ModelParameters._R[1293] := 0.75503026786797323;
stInitData.ModelParameters._R[1294] := 0.23654980202335771;
stInitData.ModelParameters._R[1295] := 0.54755224409506997;
stInitData.ModelParameters._R[1296] := 0.52533859006897188;
stInitData.ModelParameters._R[1297] := 0.90324128389400582;
stInitData.ModelParameters._R[1298] := 0.24333158147571773;
stInitData.ModelParameters._R[1299] := 0.52735687737673598;
stInitData.ModelParameters._R[1300] := 0.38713941265646878;
stInitData.ModelParameters._R[1301] := 0.89592731569932993;
stInitData.ModelParameters._R[1302] := 0.72687148834364745;
stInitData.ModelParameters._R[1303] := 0.5583773635772783;
stInitData.ModelParameters._R[1304] := 0.83005009070107882;
stInitData.ModelParameters._R[1305] := 0.4024202480847654;
stInitData.ModelParameters._R[1306] := 0.36111355814627943;
stInitData.ModelParameters._R[1307] := 0.27274668792952328;
stInitData.ModelParameters._R[1308] := 0.15128926500143677;
stInitData.ModelParameters._R[1309] := 0.23698880739223863;
stInitData.ModelParameters._R[1310] := 0.81403397584532178;
stInitData.ModelParameters._R[1311] := 0.98964549698820037;
stInitData.ModelParameters._R[1312] := 0.35552018445105205;
stInitData.ModelParameters._R[1313] := 0.53906876301218842;
stInitData.ModelParameters._R[1314] := 0.81804534396370998;
stInitData.ModelParameters._R[1315] := 0.70412084803915542;
stInitData.ModelParameters._R[1316] := 0.28763926776582305;
stInitData.ModelParameters._R[1317] := 0.76527880141033944;
stInitData.ModelParameters._R[1318] := 0.77601611998759645;
stInitData.ModelParameters._R[1319] := 0.87708295720104401;
stInitData.ModelParameters._R[1320] := 0.80341177877721182;
stInitData.ModelParameters._R[1321] := 0.75932564160319005;
stInitData.ModelParameters._R[1322] := 0.92853330194260941;
stInitData.ModelParameters._R[1323] := 0.70473832149764559;
stInitData.ModelParameters._R[1324] := 0.4047860529970061;
stInitData.ModelParameters._R[1325] := 0.7274237359401623;
stInitData.ModelParameters._R[1326] := 0.9642513942264741;
stInitData.ModelParameters._R[1327] := 0.62629828504326457;
